C09150=1155.735,302.900,-72.976,-176.899,8.332,148.732
C09151=1155.730,303.148,-73.007,-176.896,8.334,148.732
C09152=1155.726,303.397,-73.038,-176.894,8.338,148.732
C09153=1155.722,303.644,-73.070,-176.892,8.341,148.732
C09154=1155.717,303.892,-73.100,-176.889,8.344,148.732
C09155=1155.713,304.141,-73.132,-176.887,8.347,148.732
C09156=1155.709,304.389,-73.162,-176.883,8.351,148.732
C09157=1155.705,304.636,-73.193,-176.881,8.354,148.733
C09158=1155.701,304.885,-73.224,-176.878,8.357,148.733
C09159=1155.696,305.132,-73.255,-176.876,8.361,148.733
C09160=1155.692,305.381,-73.286,-176.874,8.364,148.733
C09161=1155.688,305.628,-73.318,-176.870,8.368,148.733
C09162=1155.683,305.876,-73.349,-176.868,8.371,148.733
C09163=1155.679,306.125,-73.380,-176.865,8.374,148.733
C09164=1155.675,306.373,-73.410,-176.863,8.377,148.733
C09165=1155.672,306.621,-73.442,-176.861,8.380,148.734
C09166=1155.667,306.869,-73.472,-176.858,8.383,148.733
C09167=1155.663,307.117,-73.504,-176.855,8.387,148.734
C09168=1155.659,307.365,-73.535,-176.852,8.390,148.734
C09169=1155.654,307.613,-73.566,-176.850,8.394,148.734
C09170=1155.650,307.861,-73.598,-176.848,8.397,148.734
C09171=1155.646,308.109,-73.628,-176.845,8.400,148.734
C09172=1155.642,308.357,-73.660,-176.842,8.404,148.734
C09173=1155.638,308.605,-73.691,-176.840,8.407,148.734
C09174=1155.634,308.853,-73.722,-176.837,8.410,148.734
C09175=1155.629,309.101,-73.754,-176.835,8.414,148.735
C09176=1155.625,309.349,-73.785,-176.832,8.416,148.735
C09177=1155.621,309.597,-73.816,-176.829,8.421,148.735
C09178=1155.617,309.845,-73.847,-176.827,8.424,148.735
C09179=1155.613,310.093,-73.879,-176.824,8.427,148.735
C09180=1155.609,310.341,-73.911,-176.822,8.430,148.735
C09181=1155.604,310.589,-73.941,-176.819,8.433,148.735
C09182=1155.601,310.837,-73.973,-176.816,8.437,148.735
C09183=1155.596,311.085,-74.004,-176.814,8.440,148.736
C09184=1155.592,311.333,-74.036,-176.811,8.444,148.736
C09185=1155.587,311.580,-74.068,-176.809,8.447,148.736
C09186=1155.583,311.829,-74.099,-176.806,8.451,148.736
C09187=1155.579,312.077,-74.131,-176.803,8.454,148.736
C09188=1155.575,312.325,-74.162,-176.801,8.457,148.736
C09189=1155.571,312.573,-74.194,-176.798,8.460,148.736
C09190=1155.567,312.820,-74.225,-176.796,8.464,148.736
C09191=1155.563,313.068,-74.257,-176.793,8.467,148.737
C09192=1155.558,313.346,-74.291,-176.790,8.471,148.737
C09193=1155.554,313.623,-74.327,-176.788,8.475,148.737
C09194=1155.549,313.901,-74.363,-176.784,8.478,148.737
C09195=1155.544,314.178,-74.398,-176.781,8.483,148.737
C09196=1155.540,314.426,-74.430,-176.779,8.486,148.737
C09197=1155.535,314.674,-74.461,-176.777,8.489,148.738
C09198=1155.532,314.922,-74.493,-176.774,8.492,148.738
C09199=1155.528,315.170,-74.525,-176.771,8.496,148.738
C09200=1155.523,315.418,-74.557,-176.769,8.499,148.738
C09201=1155.519,315.666,-74.589,-176.766,8.502,148.738
C09202=1155.515,315.914,-74.621,-176.764,8.506,148.738
C09203=1155.511,316.162,-74.651,-176.761,8.510,148.738
C09204=1155.506,316.410,-74.684,-176.758,8.513,148.739
C09205=1155.503,316.658,-74.716,-176.756,8.516,148.739
C09206=1155.498,316.906,-74.747,-176.753,8.519,148.739
C09207=1155.495,317.154,-74.779,-176.750,8.523,148.739
C09208=1155.490,317.402,-74.811,-176.748,8.527,148.739
C09209=1155.486,317.649,-74.843,-176.745,8.530,148.739
C09210=1155.482,317.897,-74.875,-176.743,8.533,148.739
C09211=1155.478,318.146,-74.907,-176.740,8.537,148.740
C09212=1155.473,318.393,-74.939,-176.738,8.540,148.740
C09213=1155.470,318.641,-74.970,-176.735,8.543,148.740
C09214=1155.465,318.889,-75.003,-176.733,8.547,148.740
C09215=1155.461,319.137,-75.034,-176.730,8.551,148.740
C09216=1155.457,319.385,-75.066,-176.728,8.554,148.740
C09217=1155.453,319.633,-75.099,-176.725,8.557,148.740
C09218=1155.449,319.881,-75.131,-176.723,8.560,148.741
C09219=1155.445,320.129,-75.162,-176.720,8.564,148.741
C09220=1155.441,320.376,-75.195,-176.717,8.568,148.741
C09221=1155.437,320.624,-75.227,-176.715,8.571,148.741
C09222=1155.433,320.873,-75.259,-176.712,8.575,148.741
C09223=1155.428,321.120,-75.291,-176.709,8.578,148.741
C09224=1155.425,321.368,-75.323,-176.707,8.581,148.742
C09225=1155.420,321.616,-75.355,-176.705,8.584,148.742
C09226=1155.417,321.864,-75.388,-176.702,8.589,148.742
C09227=1155.412,322.111,-75.420,-176.699,8.592,148.742
C09228=1155.408,322.359,-75.452,-176.697,8.595,148.742
C09229=1155.403,322.608,-75.484,-176.694,8.599,148.742
C09230=1155.400,322.855,-75.517,-176.692,8.602,148.743
C09231=1155.396,323.104,-75.549,-176.689,8.605,148.743
C09232=1155.391,323.351,-75.581,-176.687,8.609,148.743
C09233=1155.387,323.599,-75.613,-176.684,8.612,148.743
C09234=1155.383,323.847,-75.646,-176.681,8.616,148.743
C09235=1155.379,324.095,-75.678,-176.679,8.619,148.743
C09236=1155.375,324.343,-75.710,-176.676,8.623,148.744
C09237=1155.371,324.590,-75.743,-176.674,8.626,148.744
C09238=1155.367,324.838,-75.775,-176.672,8.630,148.744
C09239=1155.363,325.086,-75.808,-176.669,8.633,148.744
C09240=1155.359,325.334,-75.840,-176.666,8.637,148.744
C09241=1155.355,325.582,-75.872,-176.664,8.640,148.744
C09242=1155.350,325.830,-75.905,-176.661,8.643,148.745
C09243=1155.347,326.078,-75.937,-176.658,8.647,148.745
C09244=1155.342,326.325,-75.970,-176.656,8.651,148.745
C09245=1155.338,326.573,-76.002,-176.654,8.654,148.745
C09246=1155.334,326.821,-76.035,-176.651,8.658,148.745
C09247=1155.330,327.069,-76.067,-176.648,8.661,148.745
C09248=1155.326,327.317,-76.100,-176.646,8.664,148.746
C09249=1155.322,327.565,-76.132,-176.643,8.668,148.746
C09250=1155.318,327.813,-76.165,-176.641,8.672,148.746
C09251=1155.314,328.061,-76.197,-176.638,8.675,148.746
C09252=1155.309,328.308,-76.230,-176.635,8.679,148.747
C09253=1155.305,328.556,-76.262,-176.633,8.682,148.747
C09254=1155.301,328.803,-76.295,-176.631,8.686,148.747
C09255=1155.297,329.051,-76.328,-176.628,8.690,148.747
C09256=1155.293,329.300,-76.361,-176.626,8.693,148.747
C09257=1155.289,329.547,-76.394,-176.623,8.696,148.747
C09258=1155.285,329.795,-76.426,-176.620,8.700,148.748
C09259=1155.281,330.043,-76.459,-176.618,8.703,148.748
C09260=1155.277,330.291,-76.492,-176.615,8.707,148.748
C09261=1155.273,330.539,-76.525,-176.612,8.711,148.748
C09262=1155.269,330.787,-76.557,-176.610,8.714,148.748
C09263=1155.265,331.034,-76.590,-176.608,8.717,148.749
C09264=1155.261,331.282,-76.623,-176.605,8.721,148.749
C09265=1155.257,331.530,-76.656,-176.603,8.725,148.749
C09266=1155.252,331.778,-76.689,-176.600,8.728,148.749
C09267=1155.249,332.026,-76.721,-176.597,8.732,148.750
C09268=1155.245,332.273,-76.755,-176.595,8.735,148.750
C09269=1155.240,332.521,-76.788,-176.593,8.739,148.750
C09270=1155.236,332.769,-76.821,-176.590,8.743,148.750
C09271=1155.232,333.017,-76.853,-176.587,8.746,148.750
C09272=1155.228,333.265,-76.886,-176.585,8.749,148.751
C09273=1155.224,333.513,-76.920,-176.582,8.753,148.751
C09274=1155.220,333.760,-76.952,-176.580,8.757,148.751
C09275=1155.216,334.008,-76.985,-176.578,8.760,148.751
C09276=1155.212,334.255,-77.018,-176.575,8.764,148.751
C09277=1155.208,334.503,-77.052,-176.572,8.767,148.752
C09278=1155.204,334.751,-77.085,-176.570,8.771,148.752
C09279=1155.199,334.999,-77.118,-176.567,8.775,148.752
C09280=1155.195,335.246,-77.151,-176.565,8.778,148.752
C09281=1155.191,335.494,-77.184,-176.562,8.782,148.753
C09282=1155.187,335.742,-77.217,-176.560,8.785,148.753
C09283=1155.183,335.990,-77.251,-176.557,8.789,148.753
C09284=1155.179,336.237,-77.284,-176.555,8.793,148.753
C09285=1155.175,336.485,-77.317,-176.552,8.796,148.753
C09286=1155.170,336.733,-77.350,-176.549,8.800,148.754
C09287=1155.166,336.980,-77.383,-176.547,8.803,148.754
C09288=1155.163,337.229,-77.417,-176.545,8.807,148.754
C09289=1155.159,337.477,-77.450,-176.542,8.811,148.754
C09290=1155.155,337.724,-77.483,-176.539,8.814,148.755
C09291=1155.150,337.972,-77.516,-176.537,8.818,148.755
C09292=1155.146,338.220,-77.549,-176.534,8.821,148.755
C09293=1155.142,338.468,-77.582,-176.532,8.825,148.755
C09294=1155.138,338.715,-77.616,-176.529,8.829,148.755
C09295=1155.134,338.962,-77.649,-176.527,8.832,148.756
C09296=1155.130,339.243,-77.687,-176.524,8.836,148.756
C09297=1155.126,339.522,-77.725,-176.521,8.840,148.756
C09298=1155.121,339.803,-77.763,-176.518,8.844,148.756
C09299=1155.116,340.082,-77.801,-176.515,8.848,148.757
C09300=1155.112,340.330,-77.834,-176.513,8.852,148.757
C09301=1155.108,340.578,-77.867,-176.510,8.856,148.757
C09302=1155.104,340.826,-77.900,-176.508,8.859,148.757
C09303=1155.101,341.073,-77.935,-176.505,8.863,148.758
C09304=1155.096,341.321,-77.968,-176.503,8.867,148.758
C09305=1155.092,341.569,-78.002,-176.501,8.870,148.758
C09306=1155.088,341.816,-78.035,-176.498,8.874,148.758
C09307=1155.084,342.064,-78.069,-176.495,8.877,148.759
C09308=1155.079,342.312,-78.102,-176.492,8.882,148.759
C09309=1155.075,342.560,-78.137,-176.490,8.885,148.759
C09310=1155.071,342.808,-78.170,-176.487,8.889,148.759
C09311=1155.067,343.055,-78.204,-176.485,8.892,148.760
C09312=1155.063,343.302,-78.237,-176.483,8.896,148.760
C09313=1155.059,343.551,-78.271,-176.480,8.900,148.760
C09314=1155.055,343.798,-78.305,-176.478,8.903,148.760
C09315=1155.051,344.046,-78.338,-176.475,8.907,148.761
C09316=1155.047,344.293,-78.372,-176.473,8.911,148.761
C09317=1155.042,344.541,-78.406,-176.470,8.915,148.761
C09318=1155.039,344.789,-78.440,-176.467,8.918,148.761
C09319=1155.035,345.037,-78.473,-176.466,8.921,148.762
C09320=1155.030,345.284,-78.507,-176.463,8.926,148.762
C09321=1155.027,345.532,-78.542,-176.460,8.929,148.762
C09322=1155.023,345.780,-78.575,-176.457,8.933,148.762
C09323=1155.019,346.027,-78.609,-176.455,8.936,148.763
C09324=1155.014,346.275,-78.642,-176.452,8.940,148.763
C09325=1155.011,346.523,-78.677,-176.450,8.944,148.763
C09326=1155.007,346.770,-78.711,-176.447,8.948,148.764
C09327=1155.002,347.018,-78.744,-176.445,8.951,148.764
C09328=1154.999,347.266,-78.778,-176.442,8.955,148.764
C09329=1154.995,347.513,-78.813,-176.440,8.959,148.764
C09330=1154.991,347.761,-78.846,-176.438,8.962,148.764
C09331=1154.987,348.009,-78.880,-176.435,8.966,148.765
C09332=1154.983,348.256,-78.915,-176.433,8.970,148.765
C09333=1154.979,348.504,-78.948,-176.430,8.974,148.765
C09334=1154.975,348.752,-78.983,-176.428,8.977,148.766
C09335=1154.971,348.999,-79.017,-176.425,8.981,148.766
C09336=1154.966,349.246,-79.051,-176.423,8.985,148.766
C09337=1154.963,349.494,-79.085,-176.420,8.989,148.766
C09338=1154.959,349.742,-79.119,-176.418,8.992,148.767
C09339=1154.954,349.989,-79.153,-176.415,8.996,148.767
C09340=1154.951,350.237,-79.187,-176.412,8.999,148.767
C09341=1154.946,350.485,-79.222,-176.410,9.004,148.768
C09342=1154.943,350.732,-79.256,-176.408,9.007,148.768
C09343=1154.939,350.980,-79.290,-176.405,9.011,148.768
C09344=1154.935,351.227,-79.324,-176.402,9.015,148.768
C09345=1154.931,351.476,-79.358,-176.400,9.019,148.769
C09346=1154.927,351.723,-79.392,-176.398,9.022,148.769
C09347=1154.923,351.971,-79.427,-176.395,9.026,148.769
C09348=1154.918,352.218,-79.462,-176.393,9.030,148.769
C09349=1154.914,352.465,-79.495,-176.390,9.034,148.770
C09350=1154.910,352.713,-79.530,-176.388,9.037,148.770
C09351=1154.907,352.961,-79.564,-176.385,9.041,148.770
C09352=1154.903,353.209,-79.599,-176.383,9.045,148.771
C09353=1154.899,353.456,-79.633,-176.380,9.049,148.771
C09354=1154.895,353.704,-79.668,-176.378,9.052,148.771
C09355=1154.890,353.951,-79.702,-176.375,9.056,148.772
C09356=1154.887,354.199,-79.736,-176.373,9.060,148.772
C09357=1154.882,354.447,-79.771,-176.370,9.064,148.772
C09358=1154.879,354.694,-79.806,-176.368,9.067,148.772
C09359=1154.875,354.941,-79.840,-176.365,9.071,148.773
C09360=1154.871,355.189,-79.875,-176.363,9.075,148.773
C09361=1154.867,355.436,-79.909,-176.360,9.079,148.773
C09362=1154.863,355.685,-79.944,-176.358,9.082,148.774
C09363=1154.859,355.932,-79.978,-176.355,9.087,148.774
C09364=1154.855,356.180,-80.013,-176.353,9.090,148.774
C09365=1154.851,356.427,-80.048,-176.350,9.094,148.775
C09366=1154.847,356.675,-80.083,-176.348,9.098,148.775
C09367=1154.843,356.922,-80.116,-176.345,9.102,148.775
C09368=1154.839,357.170,-80.151,-176.343,9.105,148.775
C09369=1154.835,357.417,-80.186,-176.341,9.110,148.776
C09370=1154.831,357.665,-80.221,-176.338,9.113,148.776
C09371=1154.827,357.912,-80.255,-176.335,9.117,148.776
C09372=1154.824,358.159,-80.291,-176.333,9.121,148.777
C09373=1154.819,358.407,-80.325,-176.331,9.125,148.777
C09374=1154.815,358.655,-80.360,-176.328,9.129,148.777
C09375=1154.812,358.902,-80.395,-176.326,9.132,148.778
C09376=1154.808,359.150,-80.429,-176.323,9.136,148.778
C09377=1154.804,359.398,-80.464,-176.321,9.140,148.778
C09378=1154.799,359.645,-80.499,-176.318,9.144,148.779
C09379=1154.795,359.893,-80.534,-176.315,9.148,148.779
C09380=1154.792,360.140,-80.568,-176.313,9.152,148.779
C09381=1154.788,360.387,-80.604,-176.310,9.156,148.780
C09382=1154.784,360.635,-80.638,-176.308,9.159,148.780
C09383=1154.780,360.882,-80.674,-176.305,9.163,148.780
C09384=1154.776,361.130,-80.708,-176.303,9.168,148.781
C09385=1154.772,361.378,-80.744,-176.300,9.171,148.781
C09386=1154.767,361.625,-80.779,-176.297,9.175,148.781
C09387=1154.765,361.872,-80.813,-176.295,9.179,148.781
C09388=1154.761,362.121,-80.848,-176.293,9.183,148.782
C09389=1154.756,362.367,-80.883,-176.290,9.187,148.782
C09390=1154.753,362.615,-80.919,-176.287,9.191,148.782
C09391=1154.749,362.863,-80.954,-176.285,9.195,148.783
C09392=1154.744,363.110,-80.989,-176.283,9.199,148.783
C09393=1154.740,363.358,-81.024,-176.280,9.202,148.783
C09394=1154.737,363.605,-81.059,-176.278,9.207,148.784
C09395=1154.732,363.852,-81.095,-176.275,9.211,148.784
C09396=1154.729,364.100,-81.129,-176.273,9.214,148.784
C09397=1154.725,364.348,-81.165,-176.270,9.218,148.785
C09398=1154.721,364.595,-81.201,-176.267,9.223,148.785
C09399=1154.717,364.843,-81.235,-176.265,9.226,148.785
C09400=1154.713,365.126,-81.275,-176.262,9.231,148.786
C09401=1154.708,365.408,-81.316,-176.259,9.235,148.786
C09402=1154.703,365.692,-81.356,-176.257,9.240,148.787
C09403=1154.699,365.974,-81.396,-176.253,9.245,148.787
C09404=1154.696,366.222,-81.432,-176.252,9.248,148.787
C09405=1154.692,366.469,-81.467,-176.249,9.252,148.788
C09406=1154.688,366.716,-81.502,-176.246,9.257,148.788
C09407=1154.683,366.964,-81.538,-176.244,9.260,148.788
C09408=1154.679,367.212,-81.573,-176.241,9.265,148.789
C09409=1154.676,367.459,-81.609,-176.239,9.269,148.789
C09410=1154.671,367.706,-81.644,-176.237,9.272,148.790
C09411=1154.668,367.954,-81.680,-176.234,9.277,148.790
C09412=1154.664,368.201,-81.715,-176.232,9.280,148.790
C09413=1154.660,368.449,-81.751,-176.229,9.284,148.791
C09414=1154.657,368.696,-81.786,-176.227,9.289,148.791
C09415=1154.652,368.943,-81.822,-176.225,9.292,148.792
C09416=1154.648,369.191,-81.858,-176.223,9.297,148.792
C09417=1154.644,369.438,-81.893,-176.220,9.301,148.792
C09418=1154.641,369.686,-81.929,-176.218,9.304,148.793
C09419=1154.637,369.933,-81.964,-176.215,9.309,148.793
C09420=1154.633,370.180,-82.000,-176.213,9.312,148.794
C09421=1154.628,370.428,-82.036,-176.211,9.317,148.794
C09422=1154.625,370.675,-82.071,-176.208,9.321,148.795
C09423=1154.621,370.923,-82.107,-176.207,9.325,148.795
C09424=1154.617,371.170,-82.142,-176.204,9.329,148.796
C09425=1154.613,371.418,-82.178,-176.202,9.333,148.796
C09426=1154.609,371.666,-82.214,-176.200,9.337,148.796
C09427=1154.605,371.913,-82.249,-176.198,9.341,148.797
C09428=1154.601,372.160,-82.285,-176.195,9.345,148.797
C09429=1154.597,372.407,-82.322,-176.193,9.349,148.798
C09430=1154.594,372.655,-82.357,-176.191,9.353,148.798
C09431=1154.590,372.902,-82.393,-176.189,9.357,148.799
C09432=1154.586,373.150,-82.428,-176.187,9.361,148.799
C09433=1154.582,373.398,-82.464,-176.185,9.365,148.800
C09434=1154.579,373.644,-82.501,-176.183,9.369,148.800
C09435=1154.574,373.891,-82.536,-176.181,9.373,148.801
C09436=1154.570,374.139,-82.572,-176.179,9.378,148.801
C09437=1154.566,374.387,-82.608,-176.177,9.381,148.802
C09438=1154.563,374.633,-82.644,-176.175,9.385,148.802
C09439=1154.558,374.881,-82.680,-176.173,9.390,148.803
C09440=1154.555,375.129,-82.715,-176.171,9.393,148.803
C09441=1154.551,375.376,-82.751,-176.170,9.397,148.804
C09442=1154.547,375.623,-82.788,-176.167,9.401,148.804
C09443=1154.543,375.871,-82.823,-176.166,9.405,148.805
C09444=1154.539,376.118,-82.860,-176.164,9.409,148.806
C09445=1154.536,376.366,-82.896,-176.162,9.414,148.806
C09446=1154.532,376.613,-82.931,-176.160,9.418,148.807
C09447=1154.528,376.860,-82.968,-176.159,9.421,148.807
C09448=1154.524,377.108,-83.004,-176.157,9.425,148.808
C09449=1154.520,377.356,-83.040,-176.155,9.429,148.808
C09450=1154.516,377.602,-83.076,-176.154,9.433,148.809
C09451=1154.512,377.850,-83.112,-176.152,9.438,148.810
C09452=1154.509,378.097,-83.149,-176.150,9.441,148.810
C09453=1154.504,378.345,-83.185,-176.149,9.445,148.811
C09454=1154.501,378.592,-83.221,-176.148,9.449,148.812
C09455=1154.497,378.840,-83.257,-176.146,9.453,148.812
C09456=1154.493,379.087,-83.293,-176.145,9.457,148.813
C09457=1154.489,379.334,-83.330,-176.143,9.461,148.813
C09458=1154.485,379.581,-83.366,-176.142,9.465,148.814
C09459=1154.481,379.829,-83.402,-176.141,9.469,148.815
C09460=1154.478,380.076,-83.438,-176.140,9.472,148.815
C09461=1154.473,380.324,-83.474,-176.138,9.476,148.816
C09462=1154.470,380.571,-83.511,-176.137,9.480,148.817
C09463=1154.466,380.818,-83.547,-176.136,9.484,148.817
C09464=1154.462,381.065,-83.583,-176.135,9.488,148.818
C09465=1154.458,381.313,-83.620,-176.134,9.491,148.819
C09466=1154.454,381.560,-83.655,-176.133,9.496,148.820
C09467=1154.450,381.807,-83.692,-176.131,9.499,148.820
C09468=1154.447,382.054,-83.729,-176.131,9.503,148.821
C09469=1154.443,382.302,-83.765,-176.130,9.507,148.822
C09470=1154.438,382.549,-83.802,-176.129,9.510,148.822
C09471=1154.435,382.796,-83.838,-176.128,9.514,148.823
C09472=1154.431,383.044,-83.874,-176.127,9.518,148.824
C09473=1154.427,383.291,-83.910,-176.127,9.521,148.825
C09474=1154.423,383.538,-83.947,-176.126,9.525,148.825
C09475=1154.419,383.786,-83.983,-176.125,9.528,148.826
C09476=1154.415,384.033,-84.019,-176.125,9.532,148.827
C09477=1154.411,384.280,-84.056,-176.124,9.535,148.828
C09478=1154.408,384.527,-84.092,-176.123,9.539,148.828
C09479=1154.404,384.774,-84.129,-176.123,9.543,148.829
C09480=1154.400,385.022,-84.166,-176.123,9.546,148.830
C09481=1154.397,385.269,-84.202,-176.122,9.550,148.831
C09482=1154.392,385.517,-84.238,-176.122,9.553,148.832
C09483=1154.388,385.764,-84.275,-176.122,9.556,148.832
C09484=1154.385,386.011,-84.311,-176.121,9.559,148.833
C09485=1154.381,386.258,-84.348,-176.121,9.563,148.834
C09486=1154.377,386.505,-84.385,-176.121,9.566,148.835
C09487=1154.373,386.753,-84.421,-176.121,9.569,148.836
C09488=1154.369,387.000,-84.458,-176.121,9.572,148.837
C09489=1154.366,387.247,-84.494,-176.120,9.576,148.837
C09490=1154.362,387.495,-84.531,-176.121,9.579,148.838
C09491=1154.358,387.742,-84.568,-176.121,9.582,148.839
C09492=1154.354,387.990,-84.604,-176.121,9.585,148.840
C09493=1154.350,388.237,-84.640,-176.121,9.588,148.841
C09494=1154.346,388.484,-84.677,-176.121,9.591,148.842
C09495=1154.343,388.731,-84.713,-176.121,9.594,148.842
C09496=1154.339,388.978,-84.750,-176.122,9.597,148.843
C09497=1154.334,389.226,-84.786,-176.122,9.600,148.844
C09498=1154.332,389.473,-84.823,-176.122,9.603,148.845
C09499=1154.327,389.721,-84.860,-176.122,9.606,148.846
C09500=1154.323,389.968,-84.897,-176.123,9.608,148.846
C09501=1154.319,390.215,-84.934,-176.123,9.611,148.847
C09502=1154.316,390.462,-84.970,-176.124,9.614,148.848
C09503=1154.312,390.709,-85.007,-176.124,9.617,148.849
C09504=1154.307,390.996,-85.049,-176.125,9.620,148.850
C09505=1154.302,391.282,-85.091,-176.125,9.623,148.851
C09506=1154.299,391.568,-85.134,-176.125,9.626,148.852
C09507=1154.294,391.854,-85.176,-176.126,9.630,148.853
C09508=1154.291,392.102,-85.213,-176.127,9.632,148.854
C09509=1154.286,392.349,-85.250,-176.127,9.634,148.855
C09510=1154.283,392.596,-85.286,-176.128,9.637,148.855
C09511=1154.279,392.843,-85.323,-176.129,9.640,148.856
C09512=1154.275,393.090,-85.360,-176.130,9.642,148.857
C09513=1154.271,393.337,-85.397,-176.130,9.645,148.858
C09514=1154.267,393.584,-85.433,-176.130,9.647,148.859
C09515=1154.264,393.833,-85.469,-176.131,9.650,148.860
C09516=1154.260,394.080,-85.506,-176.132,9.652,148.861
C09517=1154.255,394.327,-85.543,-176.133,9.654,148.861
C09518=1154.252,394.574,-85.579,-176.133,9.657,148.862
C09519=1154.248,394.821,-85.616,-176.134,9.660,148.863
C09520=1154.244,395.068,-85.653,-176.135,9.662,148.864
C09521=1154.240,395.316,-85.690,-176.136,9.664,148.864
C09522=1154.237,395.563,-85.727,-176.136,9.667,148.865
C09523=1154.233,395.810,-85.763,-176.137,9.669,148.866
C09524=1154.229,396.058,-85.800,-176.138,9.672,148.867
C09525=1154.226,396.304,-85.836,-176.139,9.674,148.868
C09526=1154.221,396.552,-85.873,-176.140,9.675,148.869
C09527=1154.217,396.799,-85.909,-176.140,9.678,148.869
C09528=1154.213,397.047,-85.946,-176.141,9.680,148.870
C09529=1154.210,397.294,-85.983,-176.142,9.682,148.871
C09530=1154.206,397.541,-86.020,-176.142,9.685,148.872
C09531=1154.202,397.789,-86.057,-176.144,9.687,148.873
C09532=1154.198,398.036,-86.094,-176.145,9.689,148.874
C09533=1154.194,398.283,-86.130,-176.145,9.691,148.874
C09534=1154.190,398.530,-86.167,-176.146,9.693,148.875
C09535=1154.187,398.778,-86.204,-176.147,9.696,148.876
C09536=1154.183,399.025,-86.241,-176.148,9.697,148.877
C09537=1154.179,399.272,-86.278,-176.149,9.700,148.877
C09538=1154.175,399.519,-86.314,-176.150,9.702,148.878
C09539=1154.171,399.766,-86.351,-176.151,9.703,148.879
C09540=1154.167,400.013,-86.388,-176.152,9.705,148.880
C09541=1154.163,400.261,-86.424,-176.152,9.708,148.881
C09542=1154.160,400.508,-86.461,-176.153,9.710,148.881
C09543=1154.156,400.756,-86.497,-176.154,9.712,148.882
C09544=1154.152,401.003,-86.534,-176.155,9.714,148.883
C09545=1154.148,401.250,-86.571,-176.156,9.716,148.884
C09546=1154.144,401.497,-86.607,-176.157,9.718,148.884
C09547=1154.140,401.744,-86.644,-176.158,9.720,148.885
C09548=1154.137,401.992,-86.681,-176.159,9.722,148.886
C09549=1154.133,402.239,-86.718,-176.160,9.723,148.887
C09550=1154.129,402.486,-86.754,-176.161,9.726,148.887
C09551=1154.125,402.734,-86.791,-176.161,9.727,148.888
C09552=1154.121,402.981,-86.828,-176.162,9.729,148.889
C09553=1154.117,403.228,-86.865,-176.163,9.731,148.890
C09554=1154.114,403.475,-86.901,-176.164,9.733,148.890
C09555=1154.110,403.723,-86.938,-176.165,9.735,148.891
C09556=1154.106,403.970,-86.975,-176.166,9.737,148.892
C09557=1154.102,404.217,-87.012,-176.167,9.739,148.893
C09558=1154.098,404.464,-87.049,-176.167,9.740,148.893
C09559=1154.095,404.711,-87.085,-176.169,9.743,148.894
C09560=1154.091,404.958,-87.122,-176.169,9.744,148.895
C09561=1154.087,405.206,-87.159,-176.170,9.746,148.895
C09562=1154.083,405.453,-87.196,-176.171,9.748,148.896
C09563=1154.080,405.700,-87.233,-176.172,9.750,148.897
C09564=1154.076,405.947,-87.269,-176.173,9.752,148.898
C09565=1154.071,406.195,-87.306,-176.173,9.754,148.898
C09566=1154.067,406.442,-87.342,-176.174,9.755,148.899
C09567=1154.064,406.690,-87.379,-176.175,9.757,148.900
C09568=1154.060,406.937,-87.416,-176.176,9.759,148.900
C09569=1154.056,407.184,-87.453,-176.177,9.761,148.901
C09570=1154.052,407.432,-87.490,-176.178,9.763,148.902
C09571=1154.048,407.679,-87.526,-176.178,9.765,148.903
C09572=1154.045,407.926,-87.563,-176.179,9.767,148.903
C09573=1154.041,408.174,-87.600,-176.180,9.768,148.904
C09574=1154.037,408.421,-87.637,-176.181,9.770,148.904
C09575=1154.033,408.668,-87.674,-176.182,9.772,148.905
C09576=1154.029,408.915,-87.710,-176.182,9.774,148.906
C09577=1154.025,409.162,-87.747,-176.183,9.776,148.907
C09578=1154.021,409.409,-87.784,-176.183,9.778,148.907
C09579=1154.018,409.657,-87.821,-176.184,9.780,148.908
C09580=1154.014,409.904,-87.857,-176.185,9.782,148.909
C09581=1154.010,410.151,-87.894,-176.186,9.784,148.909
C09582=1154.006,410.398,-87.931,-176.186,9.785,148.910
C09583=1154.002,410.646,-87.968,-176.187,9.787,148.911
C09584=1153.998,410.893,-88.005,-176.188,9.789,148.911
C09585=1153.995,411.140,-88.041,-176.188,9.791,148.912
C09586=1153.991,411.388,-88.078,-176.189,9.792,148.913
C09587=1153.987,411.635,-88.115,-176.190,9.794,148.913
C09588=1153.983,411.882,-88.152,-176.190,9.796,148.914
C09589=1153.979,412.129,-88.189,-176.191,9.798,148.915
C09590=1153.976,412.376,-88.225,-176.192,9.799,148.915
C09591=1153.971,412.623,-88.262,-176.192,9.801,148.916
C09592=1153.968,412.871,-88.299,-176.193,9.803,148.916
C09593=1153.964,413.118,-88.336,-176.194,9.805,148.917
C09594=1153.960,413.365,-88.373,-176.195,9.807,148.918
C09595=1153.956,413.612,-88.409,-176.195,9.809,148.919
C09596=1153.952,413.860,-88.446,-176.195,9.811,148.919
C09597=1153.948,414.107,-88.483,-176.196,9.813,148.920
C09598=1153.945,414.355,-88.520,-176.197,9.814,148.920
C09599=1153.941,414.601,-88.556,-176.197,9.816,148.921
C09600=1153.937,414.849,-88.593,-176.198,9.818,148.922
C09601=1153.934,415.097,-88.630,-176.199,9.820,148.922
C09602=1153.931,415.343,-88.666,-176.199,9.821,148.923
C09603=1153.929,415.591,-88.704,-176.199,9.824,148.924
C09604=1153.928,416.003,-88.764,-176.201,9.826,148.925
C09605=1153.929,416.415,-88.824,-176.201,9.829,148.926
C09606=1153.933,416.828,-88.885,-176.202,9.832,148.927
C09607=1153.938,417.239,-88.945,-176.203,9.835,148.928
C09608=1153.517,417.241,-88.993,-176.206,9.846,148.931
C09609=1153.512,416.826,-88.932,-176.205,9.843,148.930
C09610=1153.508,416.411,-88.871,-176.204,9.841,148.929
C09611=1153.507,415.995,-88.810,-176.203,9.838,148.928
C09612=1153.509,415.578,-88.749,-176.202,9.835,148.927
C09613=1153.511,415.332,-88.712,-176.201,9.833,148.926
C09614=1153.513,415.084,-88.676,-176.201,9.831,148.926
C09615=1153.517,414.837,-88.640,-176.201,9.828,148.925
C09616=1153.520,414.589,-88.602,-176.200,9.827,148.925
C09617=1153.524,414.342,-88.565,-176.199,9.825,148.924
C09618=1153.528,414.095,-88.529,-176.199,9.824,148.923
C09619=1153.532,413.848,-88.492,-176.198,9.822,148.923
C09620=1153.536,413.601,-88.455,-176.198,9.820,148.922
C09621=1153.540,413.354,-88.419,-176.197,9.818,148.921
C09622=1153.543,413.106,-88.381,-176.196,9.816,148.921
C09623=1153.547,412.859,-88.345,-176.196,9.814,148.920
C09624=1153.551,412.612,-88.308,-176.195,9.812,148.919
C09625=1153.555,412.365,-88.271,-176.194,9.810,148.919
C09626=1153.559,412.117,-88.235,-176.194,9.808,148.918
C09627=1153.563,411.870,-88.198,-176.193,9.807,148.917
C09628=1153.566,411.623,-88.161,-176.192,9.805,148.917
C09629=1153.570,411.375,-88.124,-176.192,9.803,148.916
C09630=1153.574,411.128,-88.087,-176.191,9.801,148.915
C09631=1153.578,410.881,-88.050,-176.190,9.800,148.915
C09632=1153.582,410.634,-88.014,-176.190,9.798,148.914
C09633=1153.586,410.387,-87.977,-176.189,9.796,148.914
C09634=1153.589,410.139,-87.940,-176.188,9.794,148.913
C09635=1153.593,409.892,-87.903,-176.187,9.792,148.912
C09636=1153.597,409.645,-87.866,-176.186,9.791,148.911
C09637=1153.601,409.398,-87.830,-176.186,9.789,148.911
C09638=1153.605,409.151,-87.793,-176.185,9.787,148.910
C09639=1153.609,408.904,-87.756,-176.184,9.785,148.909
C09640=1153.612,408.656,-87.719,-176.183,9.783,148.909
C09641=1153.616,408.408,-87.682,-176.183,9.782,148.908
C09642=1153.620,408.162,-87.646,-176.182,9.780,148.907
C09643=1153.624,407.914,-87.609,-176.181,9.778,148.907
C09644=1153.628,407.667,-87.572,-176.180,9.776,148.906
C09645=1153.632,407.420,-87.536,-176.179,9.774,148.905
C09646=1153.635,407.172,-87.499,-176.179,9.772,148.905
C09647=1153.639,406.925,-87.462,-176.178,9.770,148.904
C09648=1153.643,406.678,-87.425,-176.177,9.769,148.903
C09649=1153.647,406.431,-87.388,-176.176,9.767,148.902
C09650=1153.651,406.184,-87.351,-176.175,9.765,148.902
C09651=1153.655,405.937,-87.315,-176.174,9.763,148.901
C09652=1153.658,405.689,-87.278,-176.174,9.761,148.900
C09653=1153.662,405.442,-87.241,-176.173,9.759,148.900
C09654=1153.666,405.194,-87.204,-176.172,9.758,148.899
C09655=1153.670,404.948,-87.168,-176.171,9.756,148.898
C09656=1153.674,404.700,-87.131,-176.170,9.754,148.897
C09657=1153.678,404.453,-87.094,-176.170,9.752,148.897
C09658=1153.681,404.205,-87.057,-176.168,9.750,148.896
C09659=1153.685,403.958,-87.020,-176.168,9.748,148.895
C09660=1153.689,403.711,-86.984,-176.167,9.746,148.894
C09661=1153.693,403.464,-86.947,-176.166,9.744,148.894
C09662=1153.697,403.217,-86.910,-176.165,9.742,148.893
C09663=1153.701,402.970,-86.873,-176.164,9.741,148.892
C09664=1153.704,402.722,-86.837,-176.163,9.738,148.891
C09665=1153.708,402.475,-86.800,-176.162,9.737,148.891
C09666=1153.712,402.228,-86.763,-176.161,9.735,148.890
C09667=1153.716,401.981,-86.726,-176.161,9.733,148.889
C09668=1153.719,401.734,-86.690,-176.159,9.731,148.888
C09669=1153.724,401.486,-86.653,-176.159,9.729,148.888
C09670=1153.727,401.239,-86.616,-176.158,9.727,148.887
C09671=1153.731,400.991,-86.579,-176.157,9.724,148.886
C09672=1153.735,400.744,-86.542,-176.156,9.722,148.885
C09673=1153.739,400.497,-86.507,-176.155,9.720,148.885
C09674=1153.743,400.249,-86.470,-176.155,9.719,148.884
C09675=1153.747,400.002,-86.433,-176.153,9.717,148.883
C09676=1153.751,399.754,-86.396,-176.152,9.714,148.882
C09677=1153.754,399.508,-86.359,-176.152,9.713,148.882
C09678=1153.758,399.260,-86.322,-176.151,9.711,148.881
C09679=1153.762,399.013,-86.286,-176.149,9.709,148.880
C09680=1153.766,398.766,-86.249,-176.149,9.706,148.879
C09681=1153.770,398.519,-86.212,-176.148,9.704,148.878
C09682=1153.774,398.272,-86.176,-176.147,9.702,148.878
C09683=1153.777,398.024,-86.138,-176.146,9.700,148.877
C09684=1153.781,397.777,-86.102,-176.145,9.698,148.876
C09685=1153.785,397.530,-86.065,-176.145,9.695,148.875
C09686=1153.789,397.283,-86.028,-176.144,9.693,148.874
C09687=1153.793,397.036,-85.992,-176.142,9.691,148.874
C09688=1153.797,396.788,-85.955,-176.142,9.689,148.873
C09689=1153.800,396.540,-85.917,-176.141,9.687,148.872
C09690=1153.804,396.294,-85.881,-176.140,9.684,148.871
C09691=1153.808,396.046,-85.844,-176.139,9.682,148.870
C09692=1153.812,395.799,-85.807,-176.139,9.680,148.870
C09693=1153.816,395.551,-85.771,-176.138,9.678,148.869
C09694=1153.820,395.305,-85.735,-176.137,9.675,148.868
C09695=1153.824,395.057,-85.698,-176.136,9.673,148.867
C09696=1153.827,394.809,-85.661,-176.136,9.670,148.866
C09697=1153.831,394.562,-85.624,-176.135,9.668,148.865
C09698=1153.835,394.315,-85.588,-176.134,9.665,148.865
C09699=1153.839,394.068,-85.551,-176.133,9.663,148.864
C09700=1153.843,393.821,-85.514,-176.133,9.660,148.863
C09701=1153.847,393.574,-85.477,-176.132,9.659,148.862
C09702=1153.850,393.327,-85.441,-176.131,9.656,148.861
C09703=1153.854,393.079,-85.404,-176.130,9.654,148.860
C09704=1153.858,392.832,-85.367,-176.130,9.651,148.860
C09705=1153.861,392.585,-85.331,-176.129,9.648,148.859
C09706=1153.866,392.337,-85.295,-176.129,9.645,148.858
C09707=1153.870,392.090,-85.258,-176.128,9.643,148.857
C09708=1153.874,391.843,-85.221,-176.128,9.640,148.856
C09709=1153.877,391.557,-85.178,-176.127,9.638,148.855
C09710=1153.882,391.270,-85.136,-176.126,9.635,148.854
C09711=1153.887,390.984,-85.094,-176.126,9.631,148.853
C09712=1153.891,390.698,-85.051,-176.126,9.628,148.852
C09713=1153.895,390.451,-85.014,-176.125,9.625,148.851
C09714=1153.899,390.204,-84.977,-176.124,9.622,148.851
C09715=1153.902,389.957,-84.941,-176.124,9.620,148.850
C09716=1153.907,389.709,-84.905,-176.124,9.617,148.849
C09717=1153.911,389.462,-84.868,-176.123,9.614,148.848
C09718=1153.914,389.214,-84.831,-176.123,9.611,148.847
C09719=1153.918,388.967,-84.794,-176.123,9.608,148.846
C09720=1153.922,388.720,-84.758,-176.123,9.605,148.846
C09721=1153.925,388.473,-84.721,-176.123,9.602,148.845
C09722=1153.929,388.226,-84.685,-176.122,9.600,148.844
C09723=1153.934,387.978,-84.648,-176.122,9.596,148.843
C09724=1153.937,387.731,-84.612,-176.122,9.593,148.842
C09725=1153.941,387.484,-84.575,-176.122,9.590,148.841
C09726=1153.945,387.236,-84.538,-176.122,9.587,148.841
C09727=1153.948,386.989,-84.502,-176.122,9.583,148.840
C09728=1153.952,386.741,-84.466,-176.122,9.581,148.839
C09729=1153.956,386.494,-84.429,-176.122,9.577,148.838
C09730=1153.960,386.247,-84.392,-176.123,9.574,148.837
C09731=1153.964,386.000,-84.356,-176.123,9.571,148.837
C09732=1153.968,385.753,-84.319,-176.123,9.567,148.836
C09733=1153.972,385.505,-84.283,-176.123,9.564,148.835
C09734=1153.976,385.258,-84.246,-176.124,9.561,148.834
C09735=1153.979,385.010,-84.209,-176.124,9.557,148.833
C09736=1153.983,384.763,-84.173,-176.124,9.554,148.833
C09737=1153.987,384.515,-84.137,-176.125,9.551,148.832
C09738=1153.991,384.268,-84.100,-176.125,9.547,148.831
C09739=1153.994,384.021,-84.064,-176.126,9.544,148.830
C09740=1153.999,383.774,-84.027,-176.127,9.540,148.830
C09741=1154.002,383.527,-83.991,-176.127,9.536,148.829
C09742=1154.006,383.280,-83.954,-176.128,9.533,148.828
C09743=1154.010,383.032,-83.917,-176.129,9.529,148.827
C09744=1154.014,382.785,-83.882,-176.129,9.525,148.826
C09745=1154.018,382.538,-83.845,-176.130,9.521,148.826
C09746=1154.021,382.291,-83.809,-176.131,9.518,148.825
C09747=1154.026,382.043,-83.773,-176.132,9.514,148.824
C09748=1154.030,381.796,-83.736,-176.133,9.511,148.824
C09749=1154.033,381.548,-83.699,-176.134,9.506,148.823
C09750=1154.037,381.300,-83.663,-176.135,9.503,148.822
C09751=1154.040,381.053,-83.627,-176.136,9.499,148.821
C09752=1154.045,380.806,-83.590,-176.138,9.495,148.821
C09753=1154.048,380.559,-83.554,-176.139,9.491,148.820
C09754=1154.052,380.312,-83.518,-176.140,9.488,148.819
C09755=1154.056,380.064,-83.482,-176.141,9.484,148.819
C09756=1154.060,379.817,-83.445,-176.142,9.480,148.818
C09757=1154.063,379.570,-83.409,-176.143,9.476,148.817
C09758=1154.068,379.322,-83.373,-176.145,9.472,148.817
C09759=1154.071,379.075,-83.336,-176.146,9.468,148.816
C09760=1154.076,378.828,-83.300,-176.148,9.464,148.816
C09761=1154.079,378.581,-83.264,-176.149,9.460,148.815
C09762=1154.083,378.333,-83.228,-176.150,9.456,148.814
C09763=1154.087,378.086,-83.192,-176.152,9.452,148.813
C09764=1154.091,377.838,-83.155,-176.154,9.449,148.813
C09765=1154.094,377.591,-83.119,-176.155,9.445,148.812
C09766=1154.099,377.343,-83.083,-176.157,9.440,148.812
C09767=1154.103,377.096,-83.048,-176.159,9.436,148.811
C09768=1154.107,376.849,-83.011,-176.160,9.432,148.811
C09769=1154.110,376.601,-82.975,-176.162,9.429,148.810
C09770=1154.114,376.354,-82.938,-176.164,9.424,148.809
C09771=1154.118,376.107,-82.903,-176.166,9.420,148.809
C09772=1154.122,375.860,-82.868,-176.167,9.417,148.808
C09773=1154.126,375.613,-82.831,-176.169,9.413,148.808
C09774=1154.130,375.365,-82.795,-176.171,9.408,148.807
C09775=1154.134,375.117,-82.759,-176.173,9.404,148.807
C09776=1154.138,374.870,-82.723,-176.174,9.401,148.806
C09777=1154.141,374.623,-82.687,-176.177,9.396,148.806
C09778=1154.146,374.375,-82.651,-176.179,9.393,148.805
C09779=1154.149,374.128,-82.615,-176.181,9.388,148.805
C09780=1154.153,373.881,-82.579,-176.183,9.384,148.804
C09781=1154.157,373.633,-82.543,-176.185,9.380,148.804
C09782=1154.161,373.385,-82.508,-176.187,9.376,148.803
C09783=1154.164,373.139,-82.471,-176.189,9.372,148.803
C09784=1154.169,372.891,-82.435,-176.191,9.368,148.802
C09785=1154.173,372.644,-82.400,-176.193,9.364,148.802
C09786=1154.177,372.396,-82.364,-176.195,9.360,148.801
C09787=1154.180,372.149,-82.329,-176.198,9.356,148.801
C09788=1154.184,371.902,-82.292,-176.200,9.352,148.800
C09789=1154.188,371.654,-82.256,-176.202,9.348,148.800
C09790=1154.192,371.407,-82.221,-176.204,9.344,148.799
C09791=1154.195,371.159,-82.185,-176.206,9.340,148.799
C09792=1154.200,370.912,-82.150,-176.208,9.336,148.799
C09793=1154.204,370.665,-82.114,-176.211,9.332,148.798
C09794=1154.208,370.417,-82.078,-176.213,9.327,148.798
C09795=1154.211,370.170,-82.043,-176.215,9.324,148.797
C09796=1154.216,369.922,-82.007,-176.218,9.319,148.797
C09797=1154.219,369.674,-81.971,-176.220,9.316,148.796
C09798=1154.224,369.428,-81.936,-176.222,9.311,148.796
C09799=1154.227,369.180,-81.901,-176.225,9.307,148.796
C09800=1154.231,368.932,-81.865,-176.227,9.303,148.795
C09801=1154.235,368.685,-81.829,-176.229,9.299,148.795
C09802=1154.239,368.437,-81.793,-176.231,9.296,148.794
C09803=1154.243,368.190,-81.758,-176.234,9.291,148.794
C09804=1154.247,367.943,-81.723,-176.237,9.287,148.793
C09805=1154.251,367.695,-81.687,-176.238,9.283,148.793
C09806=1154.254,367.448,-81.651,-176.241,9.279,148.793
C09807=1154.258,367.200,-81.616,-176.244,9.275,148.792
C09808=1154.262,366.954,-81.581,-176.246,9.272,148.792
C09809=1154.266,366.705,-81.546,-176.249,9.267,148.792
C09810=1154.271,366.458,-81.510,-176.251,9.263,148.791
C09811=1154.274,366.210,-81.474,-176.253,9.260,148.791
C09812=1154.279,365.963,-81.439,-176.256,9.255,148.790
C09813=1154.282,365.680,-81.399,-176.259,9.251,148.790
C09814=1154.287,365.398,-81.358,-176.262,9.246,148.790
C09815=1154.292,365.114,-81.318,-176.265,9.242,148.789
C09816=1154.296,364.832,-81.278,-176.267,9.237,148.789
C09817=1154.300,364.584,-81.243,-176.270,9.233,148.788
C09818=1154.304,364.336,-81.207,-176.273,9.229,148.788
C09819=1154.307,364.089,-81.172,-176.275,9.226,148.788
C09820=1154.312,363.841,-81.137,-176.277,9.221,148.787
C09821=1154.316,363.594,-81.102,-176.280,9.217,148.787
C09822=1154.319,363.346,-81.066,-176.282,9.213,148.787
C09823=1154.324,363.099,-81.032,-176.285,9.209,148.787
C09824=1154.327,362.851,-80.996,-176.287,9.205,148.786
C09825=1154.331,362.604,-80.961,-176.290,9.202,148.786
C09826=1154.336,362.357,-80.926,-176.293,9.198,148.786
C09827=1154.339,362.109,-80.891,-176.295,9.193,148.785
C09828=1154.343,361.861,-80.856,-176.297,9.190,148.785
C09829=1154.347,361.614,-80.821,-176.300,9.186,148.785
C09830=1154.351,361.366,-80.786,-176.302,9.182,148.784
C09831=1154.354,361.119,-80.751,-176.305,9.178,148.784
C09832=1154.359,360.871,-80.716,-176.308,9.174,148.783
C09833=1154.363,360.624,-80.681,-176.310,9.170,148.783
C09834=1154.367,360.376,-80.646,-176.313,9.166,148.783
C09835=1154.371,360.129,-80.611,-176.315,9.162,148.783
C09836=1154.374,359.881,-80.577,-176.318,9.159,148.782
C09837=1154.378,359.634,-80.541,-176.321,9.155,148.782
C09838=1154.382,359.386,-80.507,-176.322,9.151,148.782
C09839=1154.386,359.138,-80.472,-176.325,9.147,148.781
C09840=1154.391,358.891,-80.437,-176.328,9.143,148.781
C09841=1154.394,358.643,-80.402,-176.330,9.139,148.781
C09842=1154.398,358.397,-80.367,-176.333,9.135,148.780
C09843=1154.402,358.149,-80.332,-176.335,9.132,148.780
C09844=1154.407,357.901,-80.298,-176.338,9.127,148.780
C09845=1154.410,357.654,-80.262,-176.340,9.124,148.780
C09846=1154.414,357.406,-80.228,-176.343,9.120,148.779
C09847=1154.418,357.158,-80.194,-176.345,9.116,148.779
C09848=1154.422,356.910,-80.159,-176.348,9.112,148.779
C09849=1154.426,356.664,-80.124,-176.351,9.108,148.778
C09850=1154.430,356.416,-80.089,-176.353,9.105,148.778
C09851=1154.434,356.168,-80.055,-176.355,9.101,148.778
C09852=1154.438,355.920,-80.020,-176.358,9.097,148.777
C09853=1154.442,355.673,-79.986,-176.360,9.093,148.777
C09854=1154.446,355.426,-79.951,-176.363,9.090,148.777
C09855=1154.450,355.178,-79.916,-176.365,9.086,148.776
C09856=1154.453,354.930,-79.882,-176.367,9.082,148.776
C09857=1154.458,354.683,-79.848,-176.370,9.078,148.776
C09858=1154.461,354.435,-79.813,-176.373,9.075,148.776
C09859=1154.466,354.188,-79.779,-176.375,9.070,148.775
C09860=1154.470,353.940,-79.744,-176.377,9.067,148.775
C09861=1154.474,353.692,-79.710,-176.380,9.063,148.775
C09862=1154.478,353.444,-79.675,-176.383,9.059,148.774
C09863=1154.482,353.197,-79.641,-176.385,9.055,148.774
C09864=1154.485,352.949,-79.607,-176.388,9.051,148.774
C09865=1154.490,352.702,-79.571,-176.390,9.048,148.774
C09866=1154.494,352.455,-79.538,-176.393,9.044,148.773
C09867=1154.498,352.206,-79.503,-176.395,9.040,148.773
C09868=1154.502,351.959,-79.470,-176.398,9.036,148.773
C09869=1154.505,351.711,-79.435,-176.400,9.033,148.772
C09870=1154.509,351.464,-79.401,-176.403,9.029,148.772
C09871=1154.513,351.216,-79.366,-176.405,9.025,148.772
C09872=1154.517,350.969,-79.332,-176.408,9.021,148.771
C09873=1154.522,350.721,-79.298,-176.410,9.018,148.771
C09874=1154.525,350.474,-79.263,-176.413,9.014,148.771
C09875=1154.529,350.226,-79.229,-176.415,9.010,148.771
C09876=1154.533,349.978,-79.195,-176.417,9.007,148.770
C09877=1154.538,349.730,-79.161,-176.420,9.003,148.770
C09878=1154.541,349.483,-79.127,-176.423,8.999,148.770
C09879=1154.545,349.235,-79.092,-176.425,8.995,148.770
C09880=1154.549,348.988,-79.058,-176.427,8.992,148.769
C09881=1154.554,348.741,-79.024,-176.430,8.987,148.769
C09882=1154.557,348.492,-78.990,-176.433,8.984,148.769
C09883=1154.562,348.245,-78.956,-176.435,8.980,148.768
C09884=1154.566,347.998,-78.922,-176.438,8.977,148.768
C09885=1154.569,347.750,-78.888,-176.440,8.972,148.768
C09886=1154.574,347.502,-78.854,-176.442,8.969,148.768
C09887=1154.578,347.255,-78.820,-176.445,8.965,148.767
C09888=1154.582,347.007,-78.785,-176.448,8.962,148.767
C09889=1154.586,346.759,-78.752,-176.451,8.958,148.767
C09890=1154.590,346.512,-78.718,-176.452,8.954,148.766
C09891=1154.594,346.264,-78.684,-176.455,8.950,148.766
C09892=1154.598,346.016,-78.650,-176.458,8.947,148.766
C09893=1154.602,345.769,-78.617,-176.460,8.943,148.766
C09894=1154.606,345.521,-78.583,-176.463,8.939,148.766
C09895=1154.610,345.273,-78.549,-176.465,8.936,148.765
C09896=1154.613,345.026,-78.515,-176.468,8.932,148.765
C09897=1154.618,344.778,-78.481,-176.470,8.928,148.765
C09898=1154.622,344.530,-78.447,-176.473,8.924,148.764
C09899=1154.626,344.282,-78.414,-176.475,8.921,148.764
C09900=1154.630,344.035,-78.380,-176.478,8.917,148.764
C09901=1154.634,343.787,-78.346,-176.480,8.914,148.764
C09902=1154.638,343.539,-78.312,-176.483,8.910,148.764
C09903=1154.642,343.292,-78.278,-176.485,8.906,148.763
C09904=1154.646,343.044,-78.245,-176.487,8.903,148.763
C09905=1154.651,342.796,-78.211,-176.490,8.899,148.763
C09906=1154.655,342.549,-78.178,-176.493,8.895,148.762
C09907=1154.658,342.301,-78.143,-176.496,8.891,148.762
C09908=1154.662,342.053,-78.110,-176.498,8.888,148.762
C09909=1154.667,341.805,-78.077,-176.500,8.885,148.762
C09910=1154.671,341.558,-78.043,-176.503,8.881,148.762
C09911=1154.675,341.310,-78.010,-176.505,8.877,148.761
C09912=1154.678,341.062,-77.976,-176.508,8.873,148.761
C09913=1154.682,340.815,-77.942,-176.510,8.870,148.761
C09914=1154.686,340.567,-77.909,-176.513,8.865,148.760
C09915=1154.691,340.319,-77.875,-176.515,8.862,148.760
C09916=1154.695,340.072,-77.841,-176.518,8.859,148.760
C09917=1154.699,339.792,-77.803,-176.521,8.855,148.760
C09918=1154.704,339.512,-77.766,-176.524,8.851,148.760
C09919=1154.709,339.231,-77.729,-176.526,8.847,148.759
C09920=1154.713,338.951,-77.691,-176.529,8.843,148.759
C09921=1154.717,338.704,-77.657,-176.532,8.838,148.759
C09922=1154.721,338.456,-77.624,-176.535,8.835,148.759
C09923=1154.725,338.209,-77.590,-176.537,8.832,148.758
C09924=1154.730,337.961,-77.557,-176.540,8.828,148.758
C09925=1154.734,337.713,-77.524,-176.542,8.824,148.758
C09926=1154.737,337.465,-77.491,-176.544,8.820,148.757
C09927=1154.741,337.217,-77.457,-176.547,8.817,148.757
C09928=1154.745,336.970,-77.424,-176.549,8.814,148.757
C09929=1154.749,336.722,-77.390,-176.552,8.809,148.757
C09930=1154.753,336.474,-77.357,-176.554,8.806,148.757
C09931=1154.758,336.227,-77.324,-176.557,8.802,148.756
C09932=1154.762,335.979,-77.291,-176.560,8.799,148.756
C09933=1154.766,335.731,-77.258,-176.562,8.795,148.756
C09934=1154.770,335.483,-77.225,-176.565,8.791,148.756
C09935=1154.774,335.236,-77.192,-176.567,8.788,148.756
C09936=1154.778,334.988,-77.158,-176.570,8.784,148.755
C09937=1154.782,334.740,-77.125,-176.572,8.781,148.755
C09938=1154.786,334.492,-77.092,-176.575,8.777,148.755
C09939=1154.790,334.244,-77.059,-176.577,8.773,148.755
C09940=1154.794,333.996,-77.025,-176.580,8.770,148.754
C09941=1154.798,333.748,-76.994,-176.582,8.767,148.754
C09942=1154.802,333.501,-76.960,-176.585,8.763,148.754
C09943=1154.806,333.253,-76.927,-176.587,8.759,148.754
C09944=1154.810,333.005,-76.894,-176.590,8.756,148.754
C09945=1154.815,332.757,-76.861,-176.593,8.752,148.753
C09946=1154.819,332.510,-76.828,-176.595,8.749,148.753
C09947=1154.823,332.262,-76.795,-176.598,8.745,148.753
C09948=1154.827,332.014,-76.763,-176.600,8.741,148.753
C09949=1154.831,331.766,-76.730,-176.602,8.738,148.752
C09950=1154.835,331.518,-76.696,-176.605,8.734,148.752
C09951=1154.839,331.271,-76.663,-176.608,8.731,148.752
C09952=1154.843,331.022,-76.631,-176.610,8.728,148.752
C09953=1154.847,330.775,-76.598,-176.613,8.724,148.752
C09954=1154.851,330.527,-76.565,-176.616,8.720,148.752
C09955=1154.856,330.280,-76.532,-176.618,8.717,148.751
C09956=1154.860,330.032,-76.500,-176.621,8.713,148.751
C09957=1154.864,329.784,-76.467,-176.623,8.710,148.751
C09958=1154.868,329.537,-76.434,-176.625,8.706,148.751
C09959=1154.872,329.288,-76.402,-176.628,8.702,148.751
C09960=1154.876,329.041,-76.369,-176.631,8.699,148.750
C09961=1154.880,328.793,-76.335,-176.633,8.696,148.750
C09962=1154.884,328.545,-76.304,-176.636,8.692,148.750
C09963=1154.888,328.297,-76.270,-176.638,8.688,148.750
C09964=1154.893,328.049,-76.238,-176.640,8.685,148.750
C09965=1154.896,327.801,-76.205,-176.644,8.681,148.749
C09966=1154.900,327.553,-76.173,-176.646,8.678,148.749
C09967=1154.905,327.305,-76.140,-176.648,8.675,148.749
C09968=1154.909,327.059,-76.108,-176.651,8.671,148.749
C09969=1154.913,326.810,-76.075,-176.654,8.667,148.749
C09970=1154.917,326.563,-76.042,-176.656,8.664,148.748
C09971=1154.921,326.314,-76.010,-176.659,8.660,148.748
C09972=1154.925,326.066,-75.978,-176.661,8.657,148.748
C09973=1154.929,325.819,-75.945,-176.663,8.654,148.748
C09974=1154.933,325.570,-75.913,-176.667,8.650,148.748
C09975=1154.938,325.323,-75.880,-176.669,8.646,148.748
C09976=1154.942,325.075,-75.848,-176.671,8.643,148.747
C09977=1154.946,324.828,-75.815,-176.674,8.639,148.747
C09978=1154.949,324.580,-75.783,-176.677,8.636,148.747
C09979=1154.954,324.331,-75.751,-176.679,8.633,148.747
C09980=1154.957,324.084,-75.718,-176.681,8.629,148.747
C09981=1154.962,323.836,-75.686,-176.685,8.625,148.747
C09982=1154.966,323.588,-75.654,-176.687,8.622,148.746
C09983=1154.970,323.340,-75.621,-176.689,8.619,148.746
C09984=1154.974,323.092,-75.589,-176.692,8.615,148.746
C09985=1154.978,322.844,-75.557,-176.694,8.612,148.746
C09986=1154.982,322.597,-75.524,-176.697,8.608,148.746
C09987=1154.987,322.349,-75.492,-176.700,8.604,148.745
C09988=1154.991,322.101,-75.460,-176.702,8.601,148.745
C09989=1154.995,321.852,-75.428,-176.705,8.598,148.745
C09990=1154.998,321.605,-75.395,-176.707,8.595,148.745
C09991=1155.003,321.357,-75.363,-176.710,8.591,148.745
C09992=1155.007,321.109,-75.331,-176.712,8.587,148.745
C09993=1155.012,320.861,-75.299,-176.715,8.584,148.745
C09994=1155.015,320.613,-75.267,-176.718,8.580,148.744
C09995=1155.020,320.366,-75.236,-176.720,8.577,148.744
C09996=1155.024,320.118,-75.202,-176.722,8.574,148.744
//INST
///DATE 2021/06/15 17:26
///ATTR SC,RW,RJ
////FRAME ROBOT
///GROUP1 RB1
NOP
MOVL C00000 V=800.0 PL=0
MOVL C00001 V=800.0 PL=0
MOVL C00002 V=800.0 PL=0
MOVL C00003 V=800.0 PL=0
MOVL C00004 V=800.0 PL=0
MOVL C00005 V=800.0 PL=0
MOVL C00006 V=800.0 PL=0
MOVL C00007 V=800.0 PL=0
MOVL C00008 V=800.0 PL=0
MOVL C00009 V=800.0 PL=0
MOVL C00010 V=800.0 PL=0
MOVL C00011 V=800.0 PL=0
MOVL C00012 V=800.0 PL=0
MOVL C00013 V=800.0 PL=0
MOVL C00014 V=800.0 PL=0
MOVL C00015 V=800.0 PL=0
MOVL C00016 V=800.0 PL=0
MOVL C00017 V=800.0 PL=0
MOVL C00018 V=800.0 PL=0
MOVL C00019 V=800.0 PL=0
MOVL C00020 V=800.0 PL=0
MOVL C00021 V=800.0 PL=0
MOVL C00022 V=800.0 PL=0
MOVL C00023 V=800.0 PL=0
MOVL C00024 V=800.0 PL=0
MOVL C00025 V=800.0 PL=0
MOVL C00026 V=800.0 PL=0
MOVL C00027 V=800.0 PL=0
MOVL C00028 V=800.0 PL=0
MOVL C00029 V=800.0 PL=0
MOVL C00030 V=800.0 PL=0
MOVL C00031 V=800.0 PL=0
MOVL C00032 V=800.0 PL=0
MOVL C00033 V=800.0 PL=0
MOVL C00034 V=800.0 PL=0
MOVL C00035 V=800.0 PL=0
MOVL C00036 V=800.0 PL=0
MOVL C00037 V=800.0 PL=0
MOVL C00038 V=800.0 PL=0
MOVL C00039 V=800.0 PL=0
MOVL C00040 V=800.0 PL=0
MOVL C00041 V=800.0 PL=0
MOVL C00042 V=800.0 PL=0
MOVL C00043 V=800.0 PL=0
MOVL C00044 V=800.0 PL=0
MOVL C00045 V=800.0 PL=0
MOVL C00046 V=800.0 PL=0
MOVL C00047 V=800.0 PL=0
MOVL C00048 V=800.0 PL=0
MOVL C00049 V=800.0 PL=0
MOVL C00050 V=800.0 PL=0
MOVL C00051 V=800.0 PL=0
MOVL C00052 V=800.0 PL=0
MOVL C00053 V=800.0 PL=0
MOVL C00054 V=800.0 PL=0
MOVL C00055 V=800.0 PL=0
MOVL C00056 V=800.0 PL=0
MOVL C00057 V=800.0 PL=0
MOVL C00058 V=800.0 PL=0
MOVL C00059 V=800.0 PL=0
MOVL C00060 V=800.0 PL=0
MOVL C00061 V=800.0 PL=0
MOVL C00062 V=800.0 PL=0
MOVL C00063 V=800.0 PL=0
MOVL C00064 V=800.0 PL=0
MOVL C00065 V=800.0 PL=0
MOVL C00066 V=800.0 PL=0
MOVL C00067 V=800.0 PL=0
MOVL C00068 V=800.0 PL=0
MOVL C00069 V=800.0 PL=0
MOVL C00070 V=800.0 PL=0
MOVL C00071 V=800.0 PL=0
MOVL C00072 V=800.0 PL=0
MOVL C00073 V=800.0 PL=0
MOVL C00074 V=800.0 PL=0
MOVL C00075 V=800.0 PL=0
MOVL C00076 V=800.0 PL=0
MOVL C00077 V=800.0 PL=0
MOVL C00078 V=800.0 PL=0
MOVL C00079 V=800.0 PL=0
MOVL C00080 V=800.0 PL=0
MOVL C00081 V=800.0 PL=0
MOVL C00082 V=800.0 PL=0
MOVL C00083 V=800.0 PL=0
MOVL C00084 V=800.0 PL=0
MOVL C00085 V=800.0 PL=0
MOVL C00086 V=800.0 PL=0
MOVL C00087 V=800.0 PL=0
MOVL C00088 V=800.0 PL=0
MOVL C00089 V=800.0 PL=0
MOVL C00090 V=800.0 PL=0
MOVL C00091 V=800.0 PL=0
MOVL C00092 V=800.0 PL=0
MOVL C00093 V=800.0 PL=0
MOVL C00094 V=800.0 PL=0
MOVL C00095 V=800.0 PL=0
MOVL C00096 V=800.0 PL=0
MOVL C00097 V=800.0 PL=0
MOVL C00098 V=800.0 PL=0
MOVL C00099 V=800.0 PL=0
MOVL C00100 V=800.0 PL=0
MOVL C00101 V=800.0 PL=0
MOVL C00102 V=800.0 PL=0
MOVL C00103 V=800.0 PL=0
MOVL C00104 V=800.0 PL=0
MOVL C00105 V=800.0 PL=0
MOVL C00106 V=800.0 PL=0
MOVL C00107 V=800.0 PL=0
MOVL C00108 V=800.0 PL=0
MOVL C00109 V=800.0 PL=0
MOVL C00110 V=800.0 PL=0
MOVL C00111 V=800.0 PL=0
MOVL C00112 V=800.0 PL=0
MOVL C00113 V=800.0 PL=0
MOVL C00114 V=800.0 PL=0
MOVL C00115 V=800.0 PL=0
MOVL C00116 V=800.0 PL=0
MOVL C00117 V=800.0 PL=0
MOVL C00118 V=800.0 PL=0
MOVL C00119 V=800.0 PL=0
MOVL C00120 V=800.0 PL=0
MOVL C00121 V=800.0 PL=0
MOVL C00122 V=800.0 PL=0
MOVL C00123 V=800.0 PL=0
MOVL C00124 V=800.0 PL=0
MOVL C00125 V=800.0 PL=0
MOVL C00126 V=800.0 PL=0
MOVL C00127 V=800.0 PL=0
MOVL C00128 V=800.0 PL=0
MOVL C00129 V=800.0 PL=0
MOVL C00130 V=800.0 PL=0
MOVL C00131 V=800.0 PL=0
MOVL C00132 V=800.0 PL=0
MOVL C00133 V=800.0 PL=0
MOVL C00134 V=800.0 PL=0
MOVL C00135 V=800.0 PL=0
MOVL C00136 V=800.0 PL=0
MOVL C00137 V=800.0 PL=0
MOVL C00138 V=800.0 PL=0
MOVL C00139 V=800.0 PL=0
MOVL C00140 V=800.0 PL=0
MOVL C00141 V=800.0 PL=0
MOVL C00142 V=800.0 PL=0
MOVL C00143 V=800.0 PL=0
MOVL C00144 V=800.0 PL=0
MOVL C00145 V=800.0 PL=0
MOVL C00146 V=800.0 PL=0
MOVL C00147 V=800.0 PL=0
MOVL C00148 V=800.0 PL=0
MOVL C00149 V=800.0 PL=0
MOVL C00150 V=800.0 PL=0
MOVL C00151 V=800.0 PL=0
MOVL C00152 V=800.0 PL=0
MOVL C00153 V=800.0 PL=0
MOVL C00154 V=800.0 PL=0
MOVL C00155 V=800.0 PL=0
MOVL C00156 V=800.0 PL=0
MOVL C00157 V=800.0 PL=0
MOVL C00158 V=800.0 PL=0
MOVL C00159 V=800.0 PL=0
MOVL C00160 V=800.0 PL=0
MOVL C00161 V=800.0 PL=0
MOVL C00162 V=800.0 PL=0
MOVL C00163 V=800.0 PL=0
MOVL C00164 V=800.0 PL=0
MOVL C00165 V=800.0 PL=0
MOVL C00166 V=800.0 PL=0
MOVL C00167 V=800.0 PL=0
MOVL C00168 V=800.0 PL=0
MOVL C00169 V=800.0 PL=0
MOVL C00170 V=800.0 PL=0
MOVL C00171 V=800.0 PL=0
MOVL C00172 V=800.0 PL=0
MOVL C00173 V=800.0 PL=0
MOVL C00174 V=800.0 PL=0
MOVL C00175 V=800.0 PL=0
MOVL C00176 V=800.0 PL=0
MOVL C00177 V=800.0 PL=0
MOVL C00178 V=800.0 PL=0
MOVL C00179 V=800.0 PL=0
MOVL C00180 V=800.0 PL=0
MOVL C00181 V=800.0 PL=0
MOVL C00182 V=800.0 PL=0
MOVL C00183 V=800.0 PL=0
MOVL C00184 V=800.0 PL=0
MOVL C00185 V=800.0 PL=0
MOVL C00186 V=800.0 PL=0
MOVL C00187 V=800.0 PL=0
MOVL C00188 V=800.0 PL=0
MOVL C00189 V=800.0 PL=0
MOVL C00190 V=800.0 PL=0
MOVL C00191 V=800.0 PL=0
MOVL C00192 V=800.0 PL=0
MOVL C00193 V=800.0 PL=0
MOVL C00194 V=800.0 PL=0
MOVL C00195 V=800.0 PL=0
MOVL C00196 V=800.0 PL=0
MOVL C00197 V=800.0 PL=0
MOVL C00198 V=800.0 PL=0
MOVL C00199 V=800.0 PL=0
MOVL C00200 V=800.0 PL=0
MOVL C00201 V=800.0 PL=0
MOVL C00202 V=800.0 PL=0
MOVL C00203 V=800.0 PL=0
MOVL C00204 V=800.0 PL=0
MOVL C00205 V=800.0 PL=0
MOVL C00206 V=800.0 PL=0
MOVL C00207 V=800.0 PL=0
MOVL C00208 V=800.0 PL=0
MOVL C00209 V=800.0 PL=0
MOVL C00210 V=800.0 PL=0
MOVL C00211 V=800.0 PL=0
MOVL C00212 V=800.0 PL=0
MOVL C00213 V=800.0 PL=0
MOVL C00214 V=800.0 PL=0
MOVL C00215 V=800.0 PL=0
MOVL C00216 V=800.0 PL=0
MOVL C00217 V=800.0 PL=0
MOVL C00218 V=800.0 PL=0
MOVL C00219 V=800.0 PL=0
MOVL C00220 V=800.0 PL=0
MOVL C00221 V=800.0 PL=0
MOVL C00222 V=800.0 PL=0
MOVL C00223 V=800.0 PL=0
MOVL C00224 V=800.0 PL=0
MOVL C00225 V=800.0 PL=0
MOVL C00226 V=800.0 PL=0
MOVL C00227 V=800.0 PL=0
MOVL C00228 V=800.0 PL=0
MOVL C00229 V=800.0 PL=0
MOVL C00230 V=800.0 PL=0
MOVL C00231 V=800.0 PL=0
MOVL C00232 V=800.0 PL=0
MOVL C00233 V=800.0 PL=0
MOVL C00234 V=800.0 PL=0
MOVL C00235 V=800.0 PL=0
MOVL C00236 V=800.0 PL=0
MOVL C00237 V=800.0 PL=0
MOVL C00238 V=800.0 PL=0
MOVL C00239 V=800.0 PL=0
MOVL C00240 V=800.0 PL=0
MOVL C00241 V=800.0 PL=0
MOVL C00242 V=800.0 PL=0
MOVL C00243 V=800.0 PL=0
MOVL C00244 V=800.0 PL=0
MOVL C00245 V=800.0 PL=0
MOVL C00246 V=800.0 PL=0
MOVL C00247 V=800.0 PL=0
MOVL C00248 V=800.0 PL=0
MOVL C00249 V=800.0 PL=0
MOVL C00250 V=800.0 PL=0
MOVL C00251 V=800.0 PL=0
MOVL C00252 V=800.0 PL=0
MOVL C00253 V=800.0 PL=0
MOVL C00254 V=800.0 PL=0
MOVL C00255 V=800.0 PL=0
MOVL C00256 V=800.0 PL=0
MOVL C00257 V=800.0 PL=0
MOVL C00258 V=800.0 PL=0
MOVL C00259 V=800.0 PL=0
MOVL C00260 V=800.0 PL=0
MOVL C00261 V=800.0 PL=0
MOVL C00262 V=800.0 PL=0
MOVL C00263 V=800.0 PL=0
MOVL C00264 V=800.0 PL=0
MOVL C00265 V=800.0 PL=0
MOVL C00266 V=800.0 PL=0
MOVL C00267 V=800.0 PL=0
MOVL C00268 V=800.0 PL=0
MOVL C00269 V=800.0 PL=0
MOVL C00270 V=800.0 PL=0
MOVL C00271 V=800.0 PL=0
MOVL C00272 V=800.0 PL=0
MOVL C00273 V=800.0 PL=0
MOVL C00274 V=800.0 PL=0
MOVL C00275 V=800.0 PL=0
MOVL C00276 V=800.0 PL=0
MOVL C00277 V=800.0 PL=0
MOVL C00278 V=800.0 PL=0
MOVL C00279 V=800.0 PL=0
MOVL C00280 V=800.0 PL=0
MOVL C00281 V=800.0 PL=0
MOVL C00282 V=800.0 PL=0
MOVL C00283 V=800.0 PL=0
MOVL C00284 V=800.0 PL=0
MOVL C00285 V=800.0 PL=0
MOVL C00286 V=800.0 PL=0
MOVL C00287 V=800.0 PL=0
MOVL C00288 V=800.0 PL=0
MOVL C00289 V=800.0 PL=0
MOVL C00290 V=800.0 PL=0
MOVL C00291 V=800.0 PL=0
MOVL C00292 V=800.0 PL=0
MOVL C00293 V=800.0 PL=0
MOVL C00294 V=800.0 PL=0
MOVL C00295 V=800.0 PL=0
MOVL C00296 V=800.0 PL=0
MOVL C00297 V=800.0 PL=0
MOVL C00298 V=800.0 PL=0
MOVL C00299 V=800.0 PL=0
MOVL C00300 V=800.0 PL=0
MOVL C00301 V=800.0 PL=0
MOVL C00302 V=800.0 PL=0
MOVL C00303 V=800.0 PL=0
MOVL C00304 V=800.0 PL=0
MOVL C00305 V=800.0 PL=0
MOVL C00306 V=800.0 PL=0
MOVL C00307 V=800.0 PL=0
MOVL C00308 V=800.0 PL=0
MOVL C00309 V=800.0 PL=0
MOVL C00310 V=800.0 PL=0
MOVL C00311 V=800.0 PL=0
MOVL C00312 V=800.0 PL=0
MOVL C00313 V=800.0 PL=0
MOVL C00314 V=800.0 PL=0
MOVL C00315 V=800.0 PL=0
MOVL C00316 V=800.0 PL=0
MOVL C00317 V=800.0 PL=0
MOVL C00318 V=800.0 PL=0
MOVL C00319 V=800.0 PL=0
MOVL C00320 V=800.0 PL=0
MOVL C00321 V=800.0 PL=0
MOVL C00322 V=800.0 PL=0
MOVL C00323 V=800.0 PL=0
MOVL C00324 V=800.0 PL=0
MOVL C00325 V=800.0 PL=0
MOVL C00326 V=800.0 PL=0
MOVL C00327 V=800.0 PL=0
MOVL C00328 V=800.0 PL=0
MOVL C00329 V=800.0 PL=0
MOVL C00330 V=800.0 PL=0
MOVL C00331 V=800.0 PL=0
MOVL C00332 V=800.0 PL=0
MOVL C00333 V=800.0 PL=0
MOVL C00334 V=800.0 PL=0
MOVL C00335 V=800.0 PL=0
MOVL C00336 V=800.0 PL=0
MOVL C00337 V=800.0 PL=0
MOVL C00338 V=800.0 PL=0
MOVL C00339 V=800.0 PL=0
MOVL C00340 V=800.0 PL=0
MOVL C00341 V=800.0 PL=0
MOVL C00342 V=800.0 PL=0
MOVL C00343 V=800.0 PL=0
MOVL C00344 V=800.0 PL=0
MOVL C00345 V=800.0 PL=0
MOVL C00346 V=800.0 PL=0
MOVL C00347 V=800.0 PL=0
MOVL C00348 V=800.0 PL=0
MOVL C00349 V=800.0 PL=0
MOVL C00350 V=800.0 PL=0
MOVL C00351 V=800.0 PL=0
MOVL C00352 V=800.0 PL=0
MOVL C00353 V=800.0 PL=0
MOVL C00354 V=800.0 PL=0
MOVL C00355 V=800.0 PL=0
MOVL C00356 V=800.0 PL=0
MOVL C00357 V=800.0 PL=0
MOVL C00358 V=800.0 PL=0
MOVL C00359 V=800.0 PL=0
MOVL C00360 V=800.0 PL=0
MOVL C00361 V=800.0 PL=0
MOVL C00362 V=800.0 PL=0
MOVL C00363 V=800.0 PL=0
MOVL C00364 V=800.0 PL=0
MOVL C00365 V=800.0 PL=0
MOVL C00366 V=800.0 PL=0
MOVL C00367 V=800.0 PL=0
MOVL C00368 V=800.0 PL=0
MOVL C00369 V=800.0 PL=0
MOVL C00370 V=800.0 PL=0
MOVL C00371 V=800.0 PL=0
MOVL C00372 V=800.0 PL=0
MOVL C00373 V=800.0 PL=0
MOVL C00374 V=800.0 PL=0
MOVL C00375 V=800.0 PL=0
MOVL C00376 V=800.0 PL=0
MOVL C00377 V=800.0 PL=0
MOVL C00378 V=800.0 PL=0
MOVL C00379 V=800.0 PL=0
MOVL C00380 V=800.0 PL=0
MOVL C00381 V=800.0 PL=0
MOVL C00382 V=800.0 PL=0
MOVL C00383 V=800.0 PL=0
MOVL C00384 V=800.0 PL=0
MOVL C00385 V=800.0 PL=0
MOVL C00386 V=800.0 PL=0
MOVL C00387 V=800.0 PL=0
MOVL C00388 V=800.0 PL=0
MOVL C00389 V=800.0 PL=0
MOVL C00390 V=800.0 PL=0
MOVL C00391 V=800.0 PL=0
MOVL C00392 V=800.0 PL=0
MOVL C00393 V=800.0 PL=0
MOVL C00394 V=800.0 PL=0
MOVL C00395 V=800.0 PL=0
MOVL C00396 V=800.0 PL=0
MOVL C00397 V=800.0 PL=0
MOVL C00398 V=800.0 PL=0
MOVL C00399 V=800.0 PL=0
MOVL C00400 V=800.0 PL=0
MOVL C00401 V=800.0 PL=0
MOVL C00402 V=800.0 PL=0
MOVL C00403 V=800.0 PL=0
MOVL C00404 V=800.0 PL=0
MOVL C00405 V=800.0 PL=0
MOVL C00406 V=800.0 PL=0
MOVL C00407 V=800.0 PL=0
MOVL C00408 V=800.0 PL=0
MOVL C00409 V=800.0 PL=0
MOVL C00410 V=800.0 PL=0
MOVL C00411 V=800.0 PL=0
MOVL C00412 V=800.0 PL=0
MOVL C00413 V=800.0 PL=0
MOVL C00414 V=800.0 PL=0
MOVL C00415 V=800.0 PL=0
MOVL C00416 V=800.0 PL=0
MOVL C00417 V=800.0 PL=0
MOVL C00418 V=800.0 PL=0
MOVL C00419 V=800.0 PL=0
MOVL C00420 V=800.0 PL=0
MOVL C00421 V=800.0 PL=0
MOVL C00422 V=800.0 PL=0
MOVL C00423 V=800.0 PL=0
MOVL C00424 V=800.0 PL=0
MOVL C00425 V=800.0 PL=0
MOVL C00426 V=800.0 PL=0
MOVL C00427 V=800.0 PL=0
MOVL C00428 V=800.0 PL=0
MOVL C00429 V=800.0 PL=0
MOVL C00430 V=800.0 PL=0
MOVL C00431 V=800.0 PL=0
MOVL C00432 V=800.0 PL=0
MOVL C00433 V=800.0 PL=0
MOVL C00434 V=800.0 PL=0
MOVL C00435 V=800.0 PL=0
MOVL C00436 V=800.0 PL=0
MOVL C00437 V=800.0 PL=0
MOVL C00438 V=800.0 PL=0
MOVL C00439 V=800.0 PL=0
MOVL C00440 V=800.0 PL=0
MOVL C00441 V=800.0 PL=0
MOVL C00442 V=800.0 PL=0
MOVL C00443 V=800.0 PL=0
MOVL C00444 V=800.0 PL=0
MOVL C00445 V=800.0 PL=0
MOVL C00446 V=800.0 PL=0
MOVL C00447 V=800.0 PL=0
MOVL C00448 V=800.0 PL=0
MOVL C00449 V=800.0 PL=0
MOVL C00450 V=800.0 PL=0
MOVL C00451 V=800.0 PL=0
MOVL C00452 V=800.0 PL=0
MOVL C00453 V=800.0 PL=0
MOVL C00454 V=800.0 PL=0
MOVL C00455 V=800.0 PL=0
MOVL C00456 V=800.0 PL=0
MOVL C00457 V=800.0 PL=0
MOVL C00458 V=800.0 PL=0
MOVL C00459 V=800.0 PL=0
MOVL C00460 V=800.0 PL=0
MOVL C00461 V=800.0 PL=0
MOVL C00462 V=800.0 PL=0
MOVL C00463 V=800.0 PL=0
MOVL C00464 V=800.0 PL=0
MOVL C00465 V=800.0 PL=0
MOVL C00466 V=800.0 PL=0
MOVL C00467 V=800.0 PL=0
MOVL C00468 V=800.0 PL=0
MOVL C00469 V=800.0 PL=0
MOVL C00470 V=800.0 PL=0
MOVL C00471 V=800.0 PL=0
MOVL C00472 V=800.0 PL=0
MOVL C00473 V=800.0 PL=0
MOVL C00474 V=800.0 PL=0
MOVL C00475 V=800.0 PL=0
MOVL C00476 V=800.0 PL=0
MOVL C00477 V=800.0 PL=0
MOVL C00478 V=800.0 PL=0
MOVL C00479 V=800.0 PL=0
MOVL C00480 V=800.0 PL=0
MOVL C00481 V=800.0 PL=0
MOVL C00482 V=800.0 PL=0
MOVL C00483 V=800.0 PL=0
MOVL C00484 V=800.0 PL=0
MOVL C00485 V=800.0 PL=0
MOVL C00486 V=800.0 PL=0
MOVL C00487 V=800.0 PL=0
MOVL C00488 V=800.0 PL=0
MOVL C00489 V=800.0 PL=0
MOVL C00490 V=800.0 PL=0
MOVL C00491 V=800.0 PL=0
MOVL C00492 V=800.0 PL=0
MOVL C00493 V=800.0 PL=0
MOVL C00494 V=800.0 PL=0
MOVL C00495 V=800.0 PL=0
MOVL C00496 V=800.0 PL=0
MOVL C00497 V=800.0 PL=0
MOVL C00498 V=800.0 PL=0
MOVL C00499 V=800.0 PL=0
MOVL C00500 V=800.0 PL=0
MOVL C00501 V=800.0 PL=0
MOVL C00502 V=800.0 PL=0
MOVL C00503 V=800.0 PL=0
MOVL C00504 V=800.0 PL=0
MOVL C00505 V=800.0 PL=0
MOVL C00506 V=800.0 PL=0
MOVL C00507 V=800.0 PL=0
MOVL C00508 V=800.0 PL=0
MOVL C00509 V=800.0 PL=0
MOVL C00510 V=800.0 PL=0
MOVL C00511 V=800.0 PL=0
MOVL C00512 V=800.0 PL=0
MOVL C00513 V=800.0 PL=0
MOVL C00514 V=800.0 PL=0
MOVL C00515 V=800.0 PL=0
MOVL C00516 V=800.0 PL=0
MOVL C00517 V=800.0 PL=0
MOVL C00518 V=800.0 PL=0
MOVL C00519 V=800.0 PL=0
MOVL C00520 V=800.0 PL=0
MOVL C00521 V=800.0 PL=0
MOVL C00522 V=800.0 PL=0
MOVL C00523 V=800.0 PL=0
MOVL C00524 V=800.0 PL=0
MOVL C00525 V=800.0 PL=0
MOVL C00526 V=800.0 PL=0
MOVL C00527 V=800.0 PL=0
MOVL C00528 V=800.0 PL=0
MOVL C00529 V=800.0 PL=0
MOVL C00530 V=800.0 PL=0
MOVL C00531 V=800.0 PL=0
MOVL C00532 V=800.0 PL=0
MOVL C00533 V=800.0 PL=0
MOVL C00534 V=800.0 PL=0
MOVL C00535 V=800.0 PL=0
MOVL C00536 V=800.0 PL=0
MOVL C00537 V=800.0 PL=0
MOVL C00538 V=800.0 PL=0
MOVL C00539 V=800.0 PL=0
MOVL C00540 V=800.0 PL=0
MOVL C00541 V=800.0 PL=0
MOVL C00542 V=800.0 PL=0
MOVL C00543 V=800.0 PL=0
MOVL C00544 V=800.0 PL=0
MOVL C00545 V=800.0 PL=0
MOVL C00546 V=800.0 PL=0
MOVL C00547 V=800.0 PL=0
MOVL C00548 V=800.0 PL=0
MOVL C00549 V=800.0 PL=0
MOVL C00550 V=800.0 PL=0
MOVL C00551 V=800.0 PL=0
MOVL C00552 V=800.0 PL=0
MOVL C00553 V=800.0 PL=0
MOVL C00554 V=800.0 PL=0
MOVL C00555 V=800.0 PL=0
MOVL C00556 V=800.0 PL=0
MOVL C00557 V=800.0 PL=0
MOVL C00558 V=800.0 PL=0
MOVL C00559 V=800.0 PL=0
MOVL C00560 V=800.0 PL=0
MOVL C00561 V=800.0 PL=0
MOVL C00562 V=800.0 PL=0
MOVL C00563 V=800.0 PL=0
MOVL C00564 V=800.0 PL=0
MOVL C00565 V=800.0 PL=0
MOVL C00566 V=800.0 PL=0
MOVL C00567 V=800.0 PL=0
MOVL C00568 V=800.0 PL=0
MOVL C00569 V=800.0 PL=0
MOVL C00570 V=800.0 PL=0
MOVL C00571 V=800.0 PL=0
MOVL C00572 V=800.0 PL=0
MOVL C00573 V=800.0 PL=0
MOVL C00574 V=800.0 PL=0
MOVL C00575 V=800.0 PL=0
MOVL C00576 V=800.0 PL=0
MOVL C00577 V=800.0 PL=0
MOVL C00578 V=800.0 PL=0
MOVL C00579 V=800.0 PL=0
MOVL C00580 V=800.0 PL=0
MOVL C00581 V=800.0 PL=0
MOVL C00582 V=800.0 PL=0
MOVL C00583 V=800.0 PL=0
MOVL C00584 V=800.0 PL=0
MOVL C00585 V=800.0 PL=0
MOVL C00586 V=800.0 PL=0
MOVL C00587 V=800.0 PL=0
MOVL C00588 V=800.0 PL=0
MOVL C00589 V=800.0 PL=0
MOVL C00590 V=800.0 PL=0
MOVL C00591 V=800.0 PL=0
MOVL C00592 V=800.0 PL=0
MOVL C00593 V=800.0 PL=0
MOVL C00594 V=800.0 PL=0
MOVL C00595 V=800.0 PL=0
MOVL C00596 V=800.0 PL=0
MOVL C00597 V=800.0 PL=0
MOVL C00598 V=800.0 PL=0
MOVL C00599 V=800.0 PL=0
MOVL C00600 V=800.0 PL=0
MOVL C00601 V=800.0 PL=0
MOVL C00602 V=800.0 PL=0
MOVL C00603 V=800.0 PL=0
MOVL C00604 V=800.0 PL=0
MOVL C00605 V=800.0 PL=0
MOVL C00606 V=800.0 PL=0
MOVL C00607 V=800.0 PL=0
MOVL C00608 V=800.0 PL=0
MOVL C00609 V=800.0 PL=0
MOVL C00610 V=800.0 PL=0
MOVL C00611 V=800.0 PL=0
MOVL C00612 V=800.0 PL=0
MOVL C00613 V=800.0 PL=0
MOVL C00614 V=800.0 PL=0
MOVL C00615 V=800.0 PL=0
MOVL C00616 V=800.0 PL=0
MOVL C00617 V=800.0 PL=0
MOVL C00618 V=800.0 PL=0
MOVL C00619 V=800.0 PL=0
MOVL C00620 V=800.0 PL=0
MOVL C00621 V=800.0 PL=0
MOVL C00622 V=800.0 PL=0
MOVL C00623 V=800.0 PL=0
MOVL C00624 V=800.0 PL=0
MOVL C00625 V=800.0 PL=0
MOVL C00626 V=800.0 PL=0
MOVL C00627 V=800.0 PL=0
MOVL C00628 V=800.0 PL=0
MOVL C00629 V=800.0 PL=0
MOVL C00630 V=800.0 PL=0
MOVL C00631 V=800.0 PL=0
MOVL C00632 V=800.0 PL=0
MOVL C00633 V=800.0 PL=0
MOVL C00634 V=800.0 PL=0
MOVL C00635 V=800.0 PL=0
MOVL C00636 V=800.0 PL=0
MOVL C00637 V=800.0 PL=0
MOVL C00638 V=800.0 PL=0
MOVL C00639 V=800.0 PL=0
MOVL C00640 V=800.0 PL=0
MOVL C00641 V=800.0 PL=0
MOVL C00642 V=800.0 PL=0
MOVL C00643 V=800.0 PL=0
MOVL C00644 V=800.0 PL=0
MOVL C00645 V=800.0 PL=0
MOVL C00646 V=800.0 PL=0
MOVL C00647 V=800.0 PL=0
MOVL C00648 V=800.0 PL=0
MOVL C00649 V=800.0 PL=0
MOVL C00650 V=800.0 PL=0
MOVL C00651 V=800.0 PL=0
MOVL C00652 V=800.0 PL=0
MOVL C00653 V=800.0 PL=0
MOVL C00654 V=800.0 PL=0
MOVL C00655 V=800.0 PL=0
MOVL C00656 V=800.0 PL=0
MOVL C00657 V=800.0 PL=0
MOVL C00658 V=800.0 PL=0
MOVL C00659 V=800.0 PL=0
MOVL C00660 V=800.0 PL=0
MOVL C00661 V=800.0 PL=0
MOVL C00662 V=800.0 PL=0
MOVL C00663 V=800.0 PL=0
MOVL C00664 V=800.0 PL=0
MOVL C00665 V=800.0 PL=0
MOVL C00666 V=800.0 PL=0
MOVL C00667 V=800.0 PL=0
MOVL C00668 V=800.0 PL=0
MOVL C00669 V=800.0 PL=0
MOVL C00670 V=800.0 PL=0
MOVL C00671 V=800.0 PL=0
MOVL C00672 V=800.0 PL=0
MOVL C00673 V=800.0 PL=0
MOVL C00674 V=800.0 PL=0
MOVL C00675 V=800.0 PL=0
MOVL C00676 V=800.0 PL=0
MOVL C00677 V=800.0 PL=0
MOVL C00678 V=800.0 PL=0
MOVL C00679 V=800.0 PL=0
MOVL C00680 V=800.0 PL=0
MOVL C00681 V=800.0 PL=0
MOVL C00682 V=800.0 PL=0
MOVL C00683 V=800.0 PL=0
MOVL C00684 V=800.0 PL=0
MOVL C00685 V=800.0 PL=0
MOVL C00686 V=800.0 PL=0
MOVL C00687 V=800.0 PL=0
MOVL C00688 V=800.0 PL=0
MOVL C00689 V=800.0 PL=0
MOVL C00690 V=800.0 PL=0
MOVL C00691 V=800.0 PL=0
MOVL C00692 V=800.0 PL=0
MOVL C00693 V=800.0 PL=0
MOVL C00694 V=800.0 PL=0
MOVL C00695 V=800.0 PL=0
MOVL C00696 V=800.0 PL=0
MOVL C00697 V=800.0 PL=0
MOVL C00698 V=800.0 PL=0
MOVL C00699 V=800.0 PL=0
MOVL C00700 V=800.0 PL=0
MOVL C00701 V=800.0 PL=0
MOVL C00702 V=800.0 PL=0
MOVL C00703 V=800.0 PL=0
MOVL C00704 V=800.0 PL=0
MOVL C00705 V=800.0 PL=0
MOVL C00706 V=800.0 PL=0
MOVL C00707 V=800.0 PL=0
MOVL C00708 V=800.0 PL=0
MOVL C00709 V=800.0 PL=0
MOVL C00710 V=800.0 PL=0
MOVL C00711 V=800.0 PL=0
MOVL C00712 V=800.0 PL=0
MOVL C00713 V=800.0 PL=0
MOVL C00714 V=800.0 PL=0
MOVL C00715 V=800.0 PL=0
MOVL C00716 V=800.0 PL=0
MOVL C00717 V=800.0 PL=0
MOVL C00718 V=800.0 PL=0
MOVL C00719 V=800.0 PL=0
MOVL C00720 V=800.0 PL=0
MOVL C00721 V=800.0 PL=0
MOVL C00722 V=800.0 PL=0
MOVL C00723 V=800.0 PL=0
MOVL C00724 V=800.0 PL=0
MOVL C00725 V=800.0 PL=0
MOVL C00726 V=800.0 PL=0
MOVL C00727 V=800.0 PL=0
MOVL C00728 V=800.0 PL=0
MOVL C00729 V=800.0 PL=0
MOVL C00730 V=800.0 PL=0
MOVL C00731 V=800.0 PL=0
MOVL C00732 V=800.0 PL=0
MOVL C00733 V=800.0 PL=0
MOVL C00734 V=800.0 PL=0
MOVL C00735 V=800.0 PL=0
MOVL C00736 V=800.0 PL=0
MOVL C00737 V=800.0 PL=0
MOVL C00738 V=800.0 PL=0
MOVL C00739 V=800.0 PL=0
MOVL C00740 V=800.0 PL=0
MOVL C00741 V=800.0 PL=0
MOVL C00742 V=800.0 PL=0
MOVL C00743 V=800.0 PL=0
MOVL C00744 V=800.0 PL=0
MOVL C00745 V=800.0 PL=0
MOVL C00746 V=800.0 PL=0
MOVL C00747 V=800.0 PL=0
MOVL C00748 V=800.0 PL=0
MOVL C00749 V=800.0 PL=0
MOVL C00750 V=800.0 PL=0
MOVL C00751 V=800.0 PL=0
MOVL C00752 V=800.0 PL=0
MOVL C00753 V=800.0 PL=0
MOVL C00754 V=800.0 PL=0
MOVL C00755 V=800.0 PL=0
MOVL C00756 V=800.0 PL=0
MOVL C00757 V=800.0 PL=0
MOVL C00758 V=800.0 PL=0
MOVL C00759 V=800.0 PL=0
MOVL C00760 V=800.0 PL=0
MOVL C00761 V=800.0 PL=0
MOVL C00762 V=800.0 PL=0
MOVL C00763 V=800.0 PL=0
MOVL C00764 V=800.0 PL=0
MOVL C00765 V=800.0 PL=0
MOVL C00766 V=800.0 PL=0
MOVL C00767 V=800.0 PL=0
MOVL C00768 V=800.0 PL=0
MOVL C00769 V=800.0 PL=0
MOVL C00770 V=800.0 PL=0
MOVL C00771 V=800.0 PL=0
MOVL C00772 V=800.0 PL=0
MOVL C00773 V=800.0 PL=0
MOVL C00774 V=800.0 PL=0
MOVL C00775 V=800.0 PL=0
MOVL C00776 V=800.0 PL=0
MOVL C00777 V=800.0 PL=0
MOVL C00778 V=800.0 PL=0
MOVL C00779 V=800.0 PL=0
MOVL C00780 V=800.0 PL=0
MOVL C00781 V=800.0 PL=0
MOVL C00782 V=800.0 PL=0
MOVL C00783 V=800.0 PL=0
MOVL C00784 V=800.0 PL=0
MOVL C00785 V=800.0 PL=0
MOVL C00786 V=800.0 PL=0
MOVL C00787 V=800.0 PL=0
MOVL C00788 V=800.0 PL=0
MOVL C00789 V=800.0 PL=0
MOVL C00790 V=800.0 PL=0
MOVL C00791 V=800.0 PL=0
MOVL C00792 V=800.0 PL=0
MOVL C00793 V=800.0 PL=0
MOVL C00794 V=800.0 PL=0
MOVL C00795 V=800.0 PL=0
MOVL C00796 V=800.0 PL=0
MOVL C00797 V=800.0 PL=0
MOVL C00798 V=800.0 PL=0
MOVL C00799 V=800.0 PL=0
MOVL C00800 V=800.0 PL=0
MOVL C00801 V=800.0 PL=0
MOVL C00802 V=800.0 PL=0
MOVL C00803 V=800.0 PL=0
MOVL C00804 V=800.0 PL=0
MOVL C00805 V=800.0 PL=0
MOVL C00806 V=800.0 PL=0
MOVL C00807 V=800.0 PL=0
MOVL C00808 V=800.0 PL=0
MOVL C00809 V=800.0 PL=0
MOVL C00810 V=800.0 PL=0
MOVL C00811 V=800.0 PL=0
MOVL C00812 V=800.0 PL=0
MOVL C00813 V=800.0 PL=0
MOVL C00814 V=800.0 PL=0
MOVL C00815 V=800.0 PL=0
MOVL C00816 V=800.0 PL=0
MOVL C00817 V=800.0 PL=0
MOVL C00818 V=800.0 PL=0
MOVL C00819 V=800.0 PL=0
MOVL C00820 V=800.0 PL=0
MOVL C00821 V=800.0 PL=0
MOVL C00822 V=800.0 PL=0
MOVL C00823 V=800.0 PL=0
MOVL C00824 V=800.0 PL=0
MOVL C00825 V=800.0 PL=0
MOVL C00826 V=800.0 PL=0
MOVL C00827 V=800.0 PL=0
MOVL C00828 V=800.0 PL=0
MOVL C00829 V=800.0 PL=0
MOVL C00830 V=800.0 PL=0
MOVL C00831 V=800.0 PL=0
MOVL C00832 V=800.0 PL=0
MOVL C00833 V=800.0 PL=0
MOVL C00834 V=800.0 PL=0
MOVL C00835 V=800.0 PL=0
MOVL C00836 V=800.0 PL=0
MOVL C00837 V=800.0 PL=0
MOVL C00838 V=800.0 PL=0
MOVL C00839 V=800.0 PL=0
MOVL C00840 V=800.0 PL=0
MOVL C00841 V=800.0 PL=0
MOVL C00842 V=800.0 PL=0
MOVL C00843 V=800.0 PL=0
MOVL C00844 V=800.0 PL=0
MOVL C00845 V=800.0 PL=0
MOVL C00846 V=800.0 PL=0
MOVL C00847 V=800.0 PL=0
MOVL C00848 V=800.0 PL=0
MOVL C00849 V=800.0 PL=0
MOVL C00850 V=800.0 PL=0
MOVL C00851 V=800.0 PL=0
MOVL C00852 V=800.0 PL=0
MOVL C00853 V=800.0 PL=0
MOVL C00854 V=800.0 PL=0
MOVL C00855 V=800.0 PL=0
MOVL C00856 V=800.0 PL=0
MOVL C00857 V=800.0 PL=0
MOVL C00858 V=800.0 PL=0
MOVL C00859 V=800.0 PL=0
MOVL C00860 V=800.0 PL=0
MOVL C00861 V=800.0 PL=0
MOVL C00862 V=800.0 PL=0
MOVL C00863 V=800.0 PL=0
MOVL C00864 V=800.0 PL=0
MOVL C00865 V=800.0 PL=0
MOVL C00866 V=800.0 PL=0
MOVL C00867 V=800.0 PL=0
MOVL C00868 V=800.0 PL=0
MOVL C00869 V=800.0 PL=0
MOVL C00870 V=800.0 PL=0
MOVL C00871 V=800.0 PL=0
MOVL C00872 V=800.0 PL=0
MOVL C00873 V=800.0 PL=0
MOVL C00874 V=800.0 PL=0
MOVL C00875 V=800.0 PL=0
MOVL C00876 V=800.0 PL=0
MOVL C00877 V=800.0 PL=0
MOVL C00878 V=800.0 PL=0
MOVL C00879 V=800.0 PL=0
MOVL C00880 V=800.0 PL=0
MOVL C00881 V=800.0 PL=0
MOVL C00882 V=800.0 PL=0
MOVL C00883 V=800.0 PL=0
MOVL C00884 V=800.0 PL=0
MOVL C00885 V=800.0 PL=0
MOVL C00886 V=800.0 PL=0
MOVL C00887 V=800.0 PL=0
MOVL C00888 V=800.0 PL=0
MOVL C00889 V=800.0 PL=0
MOVL C00890 V=800.0 PL=0
MOVL C00891 V=800.0 PL=0
MOVL C00892 V=800.0 PL=0
MOVL C00893 V=800.0 PL=0
MOVL C00894 V=800.0 PL=0
MOVL C00895 V=800.0 PL=0
MOVL C00896 V=800.0 PL=0
MOVL C00897 V=800.0 PL=0
MOVL C00898 V=800.0 PL=0
MOVL C00899 V=800.0 PL=0
MOVL C00900 V=800.0 PL=0
MOVL C00901 V=800.0 PL=0
MOVL C00902 V=800.0 PL=0
MOVL C00903 V=800.0 PL=0
MOVL C00904 V=800.0 PL=0
MOVL C00905 V=800.0 PL=0
MOVL C00906 V=800.0 PL=0
MOVL C00907 V=800.0 PL=0
MOVL C00908 V=800.0 PL=0
MOVL C00909 V=800.0 PL=0
MOVL C00910 V=800.0 PL=0
MOVL C00911 V=800.0 PL=0
MOVL C00912 V=800.0 PL=0
MOVL C00913 V=800.0 PL=0
MOVL C00914 V=800.0 PL=0
MOVL C00915 V=800.0 PL=0
MOVL C00916 V=800.0 PL=0
MOVL C00917 V=800.0 PL=0
MOVL C00918 V=800.0 PL=0
MOVL C00919 V=800.0 PL=0
MOVL C00920 V=800.0 PL=0
MOVL C00921 V=800.0 PL=0
MOVL C00922 V=800.0 PL=0
MOVL C00923 V=800.0 PL=0
MOVL C00924 V=800.0 PL=0
MOVL C00925 V=800.0 PL=0
MOVL C00926 V=800.0 PL=0
MOVL C00927 V=800.0 PL=0
MOVL C00928 V=800.0 PL=0
MOVL C00929 V=800.0 PL=0
MOVL C00930 V=800.0 PL=0
MOVL C00931 V=800.0 PL=0
MOVL C00932 V=800.0 PL=0
MOVL C00933 V=800.0 PL=0
MOVL C00934 V=800.0 PL=0
MOVL C00935 V=800.0 PL=0
MOVL C00936 V=800.0 PL=0
MOVL C00937 V=800.0 PL=0
MOVL C00938 V=800.0 PL=0
MOVL C00939 V=800.0 PL=0
MOVL C00940 V=800.0 PL=0
MOVL C00941 V=800.0 PL=0
MOVL C00942 V=800.0 PL=0
MOVL C00943 V=800.0 PL=0
MOVL C00944 V=800.0 PL=0
MOVL C00945 V=800.0 PL=0
MOVL C00946 V=800.0 PL=0
MOVL C00947 V=800.0 PL=0
MOVL C00948 V=800.0 PL=0
MOVL C00949 V=800.0 PL=0
MOVL C00950 V=800.0 PL=0
MOVL C00951 V=800.0 PL=0
MOVL C00952 V=800.0 PL=0
MOVL C00953 V=800.0 PL=0
MOVL C00954 V=800.0 PL=0
MOVL C00955 V=800.0 PL=0
MOVL C00956 V=800.0 PL=0
MOVL C00957 V=800.0 PL=0
MOVL C00958 V=800.0 PL=0
MOVL C00959 V=800.0 PL=0
MOVL C00960 V=800.0 PL=0
MOVL C00961 V=800.0 PL=0
MOVL C00962 V=800.0 PL=0
MOVL C00963 V=800.0 PL=0
MOVL C00964 V=800.0 PL=0
MOVL C00965 V=800.0 PL=0
MOVL C00966 V=800.0 PL=0
MOVL C00967 V=800.0 PL=0
MOVL C00968 V=800.0 PL=0
MOVL C00969 V=800.0 PL=0
MOVL C00970 V=800.0 PL=0
MOVL C00971 V=800.0 PL=0
MOVL C00972 V=800.0 PL=0
MOVL C00973 V=800.0 PL=0
MOVL C00974 V=800.0 PL=0
MOVL C00975 V=800.0 PL=0
MOVL C00976 V=800.0 PL=0
MOVL C00977 V=800.0 PL=0
MOVL C00978 V=800.0 PL=0
MOVL C00979 V=800.0 PL=0
MOVL C00980 V=800.0 PL=0
MOVL C00981 V=800.0 PL=0
MOVL C00982 V=800.0 PL=0
MOVL C00983 V=800.0 PL=0
MOVL C00984 V=800.0 PL=0
MOVL C00985 V=800.0 PL=0
MOVL C00986 V=800.0 PL=0
MOVL C00987 V=800.0 PL=0
MOVL C00988 V=800.0 PL=0
MOVL C00989 V=800.0 PL=0
MOVL C00990 V=800.0 PL=0
MOVL C00991 V=800.0 PL=0
MOVL C00992 V=800.0 PL=0
MOVL C00993 V=800.0 PL=0
MOVL C00994 V=800.0 PL=0
MOVL C00995 V=800.0 PL=0
MOVL C00996 V=800.0 PL=0
MOVL C00997 V=800.0 PL=0
MOVL C00998 V=800.0 PL=0
MOVL C00999 V=800.0 PL=0
MOVL C01000 V=800.0 PL=0
MOVL C01001 V=800.0 PL=0
MOVL C01002 V=800.0 PL=0
MOVL C01003 V=800.0 PL=0
MOVL C01004 V=800.0 PL=0
MOVL C01005 V=800.0 PL=0
MOVL C01006 V=800.0 PL=0
MOVL C01007 V=800.0 PL=0
MOVL C01008 V=800.0 PL=0
MOVL C01009 V=800.0 PL=0
MOVL C01010 V=800.0 PL=0
MOVL C01011 V=800.0 PL=0
MOVL C01012 V=800.0 PL=0
MOVL C01013 V=800.0 PL=0
MOVL C01014 V=800.0 PL=0
MOVL C01015 V=800.0 PL=0
MOVL C01016 V=800.0 PL=0
MOVL C01017 V=800.0 PL=0
MOVL C01018 V=800.0 PL=0
MOVL C01019 V=800.0 PL=0
MOVL C01020 V=800.0 PL=0
MOVL C01021 V=800.0 PL=0
MOVL C01022 V=800.0 PL=0
MOVL C01023 V=800.0 PL=0
MOVL C01024 V=800.0 PL=0
MOVL C01025 V=800.0 PL=0
MOVL C01026 V=800.0 PL=0
MOVL C01027 V=800.0 PL=0
MOVL C01028 V=800.0 PL=0
MOVL C01029 V=800.0 PL=0
MOVL C01030 V=800.0 PL=0
MOVL C01031 V=800.0 PL=0
MOVL C01032 V=800.0 PL=0
MOVL C01033 V=800.0 PL=0
MOVL C01034 V=800.0 PL=0
MOVL C01035 V=800.0 PL=0
MOVL C01036 V=800.0 PL=0
MOVL C01037 V=800.0 PL=0
MOVL C01038 V=800.0 PL=0
MOVL C01039 V=800.0 PL=0
MOVL C01040 V=800.0 PL=0
MOVL C01041 V=800.0 PL=0
MOVL C01042 V=800.0 PL=0
MOVL C01043 V=800.0 PL=0
MOVL C01044 V=800.0 PL=0
MOVL C01045 V=800.0 PL=0
MOVL C01046 V=800.0 PL=0
MOVL C01047 V=800.0 PL=0
MOVL C01048 V=800.0 PL=0
MOVL C01049 V=800.0 PL=0
MOVL C01050 V=800.0 PL=0
MOVL C01051 V=800.0 PL=0
MOVL C01052 V=800.0 PL=0
MOVL C01053 V=800.0 PL=0
MOVL C01054 V=800.0 PL=0
MOVL C01055 V=800.0 PL=0
MOVL C01056 V=800.0 PL=0
MOVL C01057 V=800.0 PL=0
MOVL C01058 V=800.0 PL=0
MOVL C01059 V=800.0 PL=0
MOVL C01060 V=800.0 PL=0
MOVL C01061 V=800.0 PL=0
MOVL C01062 V=800.0 PL=0
MOVL C01063 V=800.0 PL=0
MOVL C01064 V=800.0 PL=0
MOVL C01065 V=800.0 PL=0
MOVL C01066 V=800.0 PL=0
MOVL C01067 V=800.0 PL=0
MOVL C01068 V=800.0 PL=0
MOVL C01069 V=800.0 PL=0
MOVL C01070 V=800.0 PL=0
MOVL C01071 V=800.0 PL=0
MOVL C01072 V=800.0 PL=0
MOVL C01073 V=800.0 PL=0
MOVL C01074 V=800.0 PL=0
MOVL C01075 V=800.0 PL=0
MOVL C01076 V=800.0 PL=0
MOVL C01077 V=800.0 PL=0
MOVL C01078 V=800.0 PL=0
MOVL C01079 V=800.0 PL=0
MOVL C01080 V=800.0 PL=0
MOVL C01081 V=800.0 PL=0
MOVL C01082 V=800.0 PL=0
MOVL C01083 V=800.0 PL=0
MOVL C01084 V=800.0 PL=0
MOVL C01085 V=800.0 PL=0
MOVL C01086 V=800.0 PL=0
MOVL C01087 V=800.0 PL=0
MOVL C01088 V=800.0 PL=0
MOVL C01089 V=800.0 PL=0
MOVL C01090 V=800.0 PL=0
MOVL C01091 V=800.0 PL=0
MOVL C01092 V=800.0 PL=0
MOVL C01093 V=800.0 PL=0
MOVL C01094 V=800.0 PL=0
MOVL C01095 V=800.0 PL=0
MOVL C01096 V=800.0 PL=0
MOVL C01097 V=800.0 PL=0
MOVL C01098 V=800.0 PL=0
MOVL C01099 V=800.0 PL=0
MOVL C01100 V=800.0 PL=0
MOVL C01101 V=800.0 PL=0
MOVL C01102 V=800.0 PL=0
MOVL C01103 V=800.0 PL=0
MOVL C01104 V=800.0 PL=0
MOVL C01105 V=800.0 PL=0
MOVL C01106 V=800.0 PL=0
MOVL C01107 V=800.0 PL=0
MOVL C01108 V=800.0 PL=0
MOVL C01109 V=800.0 PL=0
MOVL C01110 V=800.0 PL=0
MOVL C01111 V=800.0 PL=0
MOVL C01112 V=800.0 PL=0
MOVL C01113 V=800.0 PL=0
MOVL C01114 V=800.0 PL=0
MOVL C01115 V=800.0 PL=0
MOVL C01116 V=800.0 PL=0
MOVL C01117 V=800.0 PL=0
MOVL C01118 V=800.0 PL=0
MOVL C01119 V=800.0 PL=0
MOVL C01120 V=800.0 PL=0
MOVL C01121 V=800.0 PL=0
MOVL C01122 V=800.0 PL=0
MOVL C01123 V=800.0 PL=0
MOVL C01124 V=800.0 PL=0
MOVL C01125 V=800.0 PL=0
MOVL C01126 V=800.0 PL=0
MOVL C01127 V=800.0 PL=0
MOVL C01128 V=800.0 PL=0
MOVL C01129 V=800.0 PL=0
MOVL C01130 V=800.0 PL=0
MOVL C01131 V=800.0 PL=0
MOVL C01132 V=800.0 PL=0
MOVL C01133 V=800.0 PL=0
MOVL C01134 V=800.0 PL=0
MOVL C01135 V=800.0 PL=0
MOVL C01136 V=800.0 PL=0
MOVL C01137 V=800.0 PL=0
MOVL C01138 V=800.0 PL=0
MOVL C01139 V=800.0 PL=0
MOVL C01140 V=800.0 PL=0
MOVL C01141 V=800.0 PL=0
MOVL C01142 V=800.0 PL=0
MOVL C01143 V=800.0 PL=0
MOVL C01144 V=800.0 PL=0
MOVL C01145 V=800.0 PL=0
MOVL C01146 V=800.0 PL=0
MOVL C01147 V=800.0 PL=0
MOVL C01148 V=800.0 PL=0
MOVL C01149 V=800.0 PL=0
MOVL C01150 V=800.0 PL=0
MOVL C01151 V=800.0 PL=0
MOVL C01152 V=800.0 PL=0
MOVL C01153 V=800.0 PL=0
MOVL C01154 V=800.0 PL=0
MOVL C01155 V=800.0 PL=0
MOVL C01156 V=800.0 PL=0
MOVL C01157 V=800.0 PL=0
MOVL C01158 V=800.0 PL=0
MOVL C01159 V=800.0 PL=0
MOVL C01160 V=800.0 PL=0
MOVL C01161 V=800.0 PL=0
MOVL C01162 V=800.0 PL=0
MOVL C01163 V=800.0 PL=0
MOVL C01164 V=800.0 PL=0
MOVL C01165 V=800.0 PL=0
MOVL C01166 V=800.0 PL=0
MOVL C01167 V=800.0 PL=0
MOVL C01168 V=800.0 PL=0
MOVL C01169 V=800.0 PL=0
MOVL C01170 V=800.0 PL=0
MOVL C01171 V=800.0 PL=0
MOVL C01172 V=800.0 PL=0
MOVL C01173 V=800.0 PL=0
MOVL C01174 V=800.0 PL=0
MOVL C01175 V=800.0 PL=0
MOVL C01176 V=800.0 PL=0
MOVL C01177 V=800.0 PL=0
MOVL C01178 V=800.0 PL=0
MOVL C01179 V=800.0 PL=0
MOVL C01180 V=800.0 PL=0
MOVL C01181 V=800.0 PL=0
MOVL C01182 V=800.0 PL=0
MOVL C01183 V=800.0 PL=0
MOVL C01184 V=800.0 PL=0
MOVL C01185 V=800.0 PL=0
MOVL C01186 V=800.0 PL=0
MOVL C01187 V=800.0 PL=0
MOVL C01188 V=800.0 PL=0
MOVL C01189 V=800.0 PL=0
MOVL C01190 V=800.0 PL=0
MOVL C01191 V=800.0 PL=0
MOVL C01192 V=800.0 PL=0
MOVL C01193 V=800.0 PL=0
MOVL C01194 V=800.0 PL=0
MOVL C01195 V=800.0 PL=0
MOVL C01196 V=800.0 PL=0
MOVL C01197 V=800.0 PL=0
MOVL C01198 V=800.0 PL=0
MOVL C01199 V=800.0 PL=0
MOVL C01200 V=800.0 PL=0
MOVL C01201 V=800.0 PL=0
MOVL C01202 V=800.0 PL=0
MOVL C01203 V=800.0 PL=0
MOVL C01204 V=800.0 PL=0
MOVL C01205 V=800.0 PL=0
MOVL C01206 V=800.0 PL=0
MOVL C01207 V=800.0 PL=0
MOVL C01208 V=800.0 PL=0
MOVL C01209 V=800.0 PL=0
MOVL C01210 V=800.0 PL=0
MOVL C01211 V=800.0 PL=0
MOVL C01212 V=800.0 PL=0
MOVL C01213 V=800.0 PL=0
MOVL C01214 V=800.0 PL=0
MOVL C01215 V=800.0 PL=0
MOVL C01216 V=800.0 PL=0
MOVL C01217 V=800.0 PL=0
MOVL C01218 V=800.0 PL=0
MOVL C01219 V=800.0 PL=0
MOVL C01220 V=800.0 PL=0
MOVL C01221 V=800.0 PL=0
MOVL C01222 V=800.0 PL=0
MOVL C01223 V=800.0 PL=0
MOVL C01224 V=800.0 PL=0
MOVL C01225 V=800.0 PL=0
MOVL C01226 V=800.0 PL=0
MOVL C01227 V=800.0 PL=0
MOVL C01228 V=800.0 PL=0
MOVL C01229 V=800.0 PL=0
MOVL C01230 V=800.0 PL=0
MOVL C01231 V=800.0 PL=0
MOVL C01232 V=800.0 PL=0
MOVL C01233 V=800.0 PL=0
MOVL C01234 V=800.0 PL=0
MOVL C01235 V=800.0 PL=0
MOVL C01236 V=800.0 PL=0
MOVL C01237 V=800.0 PL=0
MOVL C01238 V=800.0 PL=0
MOVL C01239 V=800.0 PL=0
MOVL C01240 V=800.0 PL=0
MOVL C01241 V=800.0 PL=0
MOVL C01242 V=800.0 PL=0
MOVL C01243 V=800.0 PL=0
MOVL C01244 V=800.0 PL=0
MOVL C01245 V=800.0 PL=0
MOVL C01246 V=800.0 PL=0
MOVL C01247 V=800.0 PL=0
MOVL C01248 V=800.0 PL=0
MOVL C01249 V=800.0 PL=0
MOVL C01250 V=800.0 PL=0
MOVL C01251 V=800.0 PL=0
MOVL C01252 V=800.0 PL=0
MOVL C01253 V=800.0 PL=0
MOVL C01254 V=800.0 PL=0
MOVL C01255 V=800.0 PL=0
MOVL C01256 V=800.0 PL=0
MOVL C01257 V=800.0 PL=0
MOVL C01258 V=800.0 PL=0
MOVL C01259 V=800.0 PL=0
MOVL C01260 V=800.0 PL=0
MOVL C01261 V=800.0 PL=0
MOVL C01262 V=800.0 PL=0
MOVL C01263 V=800.0 PL=0
MOVL C01264 V=800.0 PL=0
MOVL C01265 V=800.0 PL=0
MOVL C01266 V=800.0 PL=0
MOVL C01267 V=800.0 PL=0
MOVL C01268 V=800.0 PL=0
MOVL C01269 V=800.0 PL=0
MOVL C01270 V=800.0 PL=0
MOVL C01271 V=800.0 PL=0
MOVL C01272 V=800.0 PL=0
MOVL C01273 V=800.0 PL=0
MOVL C01274 V=800.0 PL=0
MOVL C01275 V=800.0 PL=0
MOVL C01276 V=800.0 PL=0
MOVL C01277 V=800.0 PL=0
MOVL C01278 V=800.0 PL=0
MOVL C01279 V=800.0 PL=0
MOVL C01280 V=800.0 PL=0
MOVL C01281 V=800.0 PL=0
MOVL C01282 V=800.0 PL=0
MOVL C01283 V=800.0 PL=0
MOVL C01284 V=800.0 PL=0
MOVL C01285 V=800.0 PL=0
MOVL C01286 V=800.0 PL=0
MOVL C01287 V=800.0 PL=0
MOVL C01288 V=800.0 PL=0
MOVL C01289 V=800.0 PL=0
MOVL C01290 V=800.0 PL=0
MOVL C01291 V=800.0 PL=0
MOVL C01292 V=800.0 PL=0
MOVL C01293 V=800.0 PL=0
MOVL C01294 V=800.0 PL=0
MOVL C01295 V=800.0 PL=0
MOVL C01296 V=800.0 PL=0
MOVL C01297 V=800.0 PL=0
MOVL C01298 V=800.0 PL=0
MOVL C01299 V=800.0 PL=0
MOVL C01300 V=800.0 PL=0
MOVL C01301 V=800.0 PL=0
MOVL C01302 V=800.0 PL=0
MOVL C01303 V=800.0 PL=0
MOVL C01304 V=800.0 PL=0
MOVL C01305 V=800.0 PL=0
MOVL C01306 V=800.0 PL=0
MOVL C01307 V=800.0 PL=0
MOVL C01308 V=800.0 PL=0
MOVL C01309 V=800.0 PL=0
MOVL C01310 V=800.0 PL=0
MOVL C01311 V=800.0 PL=0
MOVL C01312 V=800.0 PL=0
MOVL C01313 V=800.0 PL=0
MOVL C01314 V=800.0 PL=0
MOVL C01315 V=800.0 PL=0
MOVL C01316 V=800.0 PL=0
MOVL C01317 V=800.0 PL=0
MOVL C01318 V=800.0 PL=0
MOVL C01319 V=800.0 PL=0
MOVL C01320 V=800.0 PL=0
MOVL C01321 V=800.0 PL=0
MOVL C01322 V=800.0 PL=0
MOVL C01323 V=800.0 PL=0
MOVL C01324 V=800.0 PL=0
MOVL C01325 V=800.0 PL=0
MOVL C01326 V=800.0 PL=0
MOVL C01327 V=800.0 PL=0
MOVL C01328 V=800.0 PL=0
MOVL C01329 V=800.0 PL=0
MOVL C01330 V=800.0 PL=0
MOVL C01331 V=800.0 PL=0
MOVL C01332 V=800.0 PL=0
MOVL C01333 V=800.0 PL=0
MOVL C01334 V=800.0 PL=0
MOVL C01335 V=800.0 PL=0
MOVL C01336 V=800.0 PL=0
MOVL C01337 V=800.0 PL=0
MOVL C01338 V=800.0 PL=0
MOVL C01339 V=800.0 PL=0
MOVL C01340 V=800.0 PL=0
MOVL C01341 V=800.0 PL=0
MOVL C01342 V=800.0 PL=0
MOVL C01343 V=800.0 PL=0
MOVL C01344 V=800.0 PL=0
MOVL C01345 V=800.0 PL=0
MOVL C01346 V=800.0 PL=0
MOVL C01347 V=800.0 PL=0
MOVL C01348 V=800.0 PL=0
MOVL C01349 V=800.0 PL=0
MOVL C01350 V=800.0 PL=0
MOVL C01351 V=800.0 PL=0
MOVL C01352 V=800.0 PL=0
MOVL C01353 V=800.0 PL=0
MOVL C01354 V=800.0 PL=0
MOVL C01355 V=800.0 PL=0
MOVL C01356 V=800.0 PL=0
MOVL C01357 V=800.0 PL=0
MOVL C01358 V=800.0 PL=0
MOVL C01359 V=800.0 PL=0
MOVL C01360 V=800.0 PL=0
MOVL C01361 V=800.0 PL=0
MOVL C01362 V=800.0 PL=0
MOVL C01363 V=800.0 PL=0
MOVL C01364 V=800.0 PL=0
MOVL C01365 V=800.0 PL=0
MOVL C01366 V=800.0 PL=0
MOVL C01367 V=800.0 PL=0
MOVL C01368 V=800.0 PL=0
MOVL C01369 V=800.0 PL=0
MOVL C01370 V=800.0 PL=0
MOVL C01371 V=800.0 PL=0
MOVL C01372 V=800.0 PL=0
MOVL C01373 V=800.0 PL=0
MOVL C01374 V=800.0 PL=0
MOVL C01375 V=800.0 PL=0
MOVL C01376 V=800.0 PL=0
MOVL C01377 V=800.0 PL=0
MOVL C01378 V=800.0 PL=0
MOVL C01379 V=800.0 PL=0
MOVL C01380 V=800.0 PL=0
MOVL C01381 V=800.0 PL=0
MOVL C01382 V=800.0 PL=0
MOVL C01383 V=800.0 PL=0
MOVL C01384 V=800.0 PL=0
MOVL C01385 V=800.0 PL=0
MOVL C01386 V=800.0 PL=0
MOVL C01387 V=800.0 PL=0
MOVL C01388 V=800.0 PL=0
MOVL C01389 V=800.0 PL=0
MOVL C01390 V=800.0 PL=0
MOVL C01391 V=800.0 PL=0
MOVL C01392 V=800.0 PL=0
MOVL C01393 V=800.0 PL=0
MOVL C01394 V=800.0 PL=0
MOVL C01395 V=800.0 PL=0
MOVL C01396 V=800.0 PL=0
MOVL C01397 V=800.0 PL=0
MOVL C01398 V=800.0 PL=0
MOVL C01399 V=800.0 PL=0
MOVL C01400 V=800.0 PL=0
MOVL C01401 V=800.0 PL=0
MOVL C01402 V=800.0 PL=0
MOVL C01403 V=800.0 PL=0
MOVL C01404 V=800.0 PL=0
MOVL C01405 V=800.0 PL=0
MOVL C01406 V=800.0 PL=0
MOVL C01407 V=800.0 PL=0
MOVL C01408 V=800.0 PL=0
MOVL C01409 V=800.0 PL=0
MOVL C01410 V=800.0 PL=0
MOVL C01411 V=800.0 PL=0
MOVL C01412 V=800.0 PL=0
MOVL C01413 V=800.0 PL=0
MOVL C01414 V=800.0 PL=0
MOVL C01415 V=800.0 PL=0
MOVL C01416 V=800.0 PL=0
MOVL C01417 V=800.0 PL=0
MOVL C01418 V=800.0 PL=0
MOVL C01419 V=800.0 PL=0
MOVL C01420 V=800.0 PL=0
MOVL C01421 V=800.0 PL=0
MOVL C01422 V=800.0 PL=0
MOVL C01423 V=800.0 PL=0
MOVL C01424 V=800.0 PL=0
MOVL C01425 V=800.0 PL=0
MOVL C01426 V=800.0 PL=0
MOVL C01427 V=800.0 PL=0
MOVL C01428 V=800.0 PL=0
MOVL C01429 V=800.0 PL=0
MOVL C01430 V=800.0 PL=0
MOVL C01431 V=800.0 PL=0
MOVL C01432 V=800.0 PL=0
MOVL C01433 V=800.0 PL=0
MOVL C01434 V=800.0 PL=0
MOVL C01435 V=800.0 PL=0
MOVL C01436 V=800.0 PL=0
MOVL C01437 V=800.0 PL=0
MOVL C01438 V=800.0 PL=0
MOVL C01439 V=800.0 PL=0
MOVL C01440 V=800.0 PL=0
MOVL C01441 V=800.0 PL=0
MOVL C01442 V=800.0 PL=0
MOVL C01443 V=800.0 PL=0
MOVL C01444 V=800.0 PL=0
MOVL C01445 V=800.0 PL=0
MOVL C01446 V=800.0 PL=0
MOVL C01447 V=800.0 PL=0
MOVL C01448 V=800.0 PL=0
MOVL C01449 V=800.0 PL=0
MOVL C01450 V=800.0 PL=0
MOVL C01451 V=800.0 PL=0
MOVL C01452 V=800.0 PL=0
MOVL C01453 V=800.0 PL=0
MOVL C01454 V=800.0 PL=0
MOVL C01455 V=800.0 PL=0
MOVL C01456 V=800.0 PL=0
MOVL C01457 V=800.0 PL=0
MOVL C01458 V=800.0 PL=0
MOVL C01459 V=800.0 PL=0
MOVL C01460 V=800.0 PL=0
MOVL C01461 V=800.0 PL=0
MOVL C01462 V=800.0 PL=0
MOVL C01463 V=800.0 PL=0
MOVL C01464 V=800.0 PL=0
MOVL C01465 V=800.0 PL=0
MOVL C01466 V=800.0 PL=0
MOVL C01467 V=800.0 PL=0
MOVL C01468 V=800.0 PL=0
MOVL C01469 V=800.0 PL=0
MOVL C01470 V=800.0 PL=0
MOVL C01471 V=800.0 PL=0
MOVL C01472 V=800.0 PL=0
MOVL C01473 V=800.0 PL=0
MOVL C01474 V=800.0 PL=0
MOVL C01475 V=800.0 PL=0
MOVL C01476 V=800.0 PL=0
MOVL C01477 V=800.0 PL=0
MOVL C01478 V=800.0 PL=0
MOVL C01479 V=800.0 PL=0
MOVL C01480 V=800.0 PL=0
MOVL C01481 V=800.0 PL=0
MOVL C01482 V=800.0 PL=0
MOVL C01483 V=800.0 PL=0
MOVL C01484 V=800.0 PL=0
MOVL C01485 V=800.0 PL=0
MOVL C01486 V=800.0 PL=0
MOVL C01487 V=800.0 PL=0
MOVL C01488 V=800.0 PL=0
MOVL C01489 V=800.0 PL=0
MOVL C01490 V=800.0 PL=0
MOVL C01491 V=800.0 PL=0
MOVL C01492 V=800.0 PL=0
MOVL C01493 V=800.0 PL=0
MOVL C01494 V=800.0 PL=0
MOVL C01495 V=800.0 PL=0
MOVL C01496 V=800.0 PL=0
MOVL C01497 V=800.0 PL=0
MOVL C01498 V=800.0 PL=0
MOVL C01499 V=800.0 PL=0
MOVL C01500 V=800.0 PL=0
MOVL C01501 V=800.0 PL=0
MOVL C01502 V=800.0 PL=0
MOVL C01503 V=800.0 PL=0
MOVL C01504 V=800.0 PL=0
MOVL C01505 V=800.0 PL=0
MOVL C01506 V=800.0 PL=0
MOVL C01507 V=800.0 PL=0
MOVL C01508 V=800.0 PL=0
MOVL C01509 V=800.0 PL=0
MOVL C01510 V=800.0 PL=0
MOVL C01511 V=800.0 PL=0
MOVL C01512 V=800.0 PL=0
MOVL C01513 V=800.0 PL=0
MOVL C01514 V=800.0 PL=0
MOVL C01515 V=800.0 PL=0
MOVL C01516 V=800.0 PL=0
MOVL C01517 V=800.0 PL=0
MOVL C01518 V=800.0 PL=0
MOVL C01519 V=800.0 PL=0
MOVL C01520 V=800.0 PL=0
MOVL C01521 V=800.0 PL=0
MOVL C01522 V=800.0 PL=0
MOVL C01523 V=800.0 PL=0
MOVL C01524 V=800.0 PL=0
MOVL C01525 V=800.0 PL=0
MOVL C01526 V=800.0 PL=0
MOVL C01527 V=800.0 PL=0
MOVL C01528 V=800.0 PL=0
MOVL C01529 V=800.0 PL=0
MOVL C01530 V=800.0 PL=0
MOVL C01531 V=800.0 PL=0
MOVL C01532 V=800.0 PL=0
MOVL C01533 V=800.0 PL=0
MOVL C01534 V=800.0 PL=0
MOVL C01535 V=800.0 PL=0
MOVL C01536 V=800.0 PL=0
MOVL C01537 V=800.0 PL=0
MOVL C01538 V=800.0 PL=0
MOVL C01539 V=800.0 PL=0
MOVL C01540 V=800.0 PL=0
MOVL C01541 V=800.0 PL=0
MOVL C01542 V=800.0 PL=0
MOVL C01543 V=800.0 PL=0
MOVL C01544 V=800.0 PL=0
MOVL C01545 V=800.0 PL=0
MOVL C01546 V=800.0 PL=0
MOVL C01547 V=800.0 PL=0
MOVL C01548 V=800.0 PL=0
MOVL C01549 V=800.0 PL=0
MOVL C01550 V=800.0 PL=0
MOVL C01551 V=800.0 PL=0
MOVL C01552 V=800.0 PL=0
MOVL C01553 V=800.0 PL=0
MOVL C01554 V=800.0 PL=0
MOVL C01555 V=800.0 PL=0
MOVL C01556 V=800.0 PL=0
MOVL C01557 V=800.0 PL=0
MOVL C01558 V=800.0 PL=0
MOVL C01559 V=800.0 PL=0
MOVL C01560 V=800.0 PL=0
MOVL C01561 V=800.0 PL=0
MOVL C01562 V=800.0 PL=0
MOVL C01563 V=800.0 PL=0
MOVL C01564 V=800.0 PL=0
MOVL C01565 V=800.0 PL=0
MOVL C01566 V=800.0 PL=0
MOVL C01567 V=800.0 PL=0
MOVL C01568 V=800.0 PL=0
MOVL C01569 V=800.0 PL=0
MOVL C01570 V=800.0 PL=0
MOVL C01571 V=800.0 PL=0
MOVL C01572 V=800.0 PL=0
MOVL C01573 V=800.0 PL=0
MOVL C01574 V=800.0 PL=0
MOVL C01575 V=800.0 PL=0
MOVL C01576 V=800.0 PL=0
MOVL C01577 V=800.0 PL=0
MOVL C01578 V=800.0 PL=0
MOVL C01579 V=800.0 PL=0
MOVL C01580 V=800.0 PL=0
MOVL C01581 V=800.0 PL=0
MOVL C01582 V=800.0 PL=0
MOVL C01583 V=800.0 PL=0
MOVL C01584 V=800.0 PL=0
MOVL C01585 V=800.0 PL=0
MOVL C01586 V=800.0 PL=0
MOVL C01587 V=800.0 PL=0
MOVL C01588 V=800.0 PL=0
MOVL C01589 V=800.0 PL=0
MOVL C01590 V=800.0 PL=0
MOVL C01591 V=800.0 PL=0
MOVL C01592 V=800.0 PL=0
MOVL C01593 V=800.0 PL=0
MOVL C01594 V=800.0 PL=0
MOVL C01595 V=800.0 PL=0
MOVL C01596 V=800.0 PL=0
MOVL C01597 V=800.0 PL=0
MOVL C01598 V=800.0 PL=0
MOVL C01599 V=800.0 PL=0
MOVL C01600 V=800.0 PL=0
MOVL C01601 V=800.0 PL=0
MOVL C01602 V=800.0 PL=0
MOVL C01603 V=800.0 PL=0
MOVL C01604 V=800.0 PL=0
MOVL C01605 V=800.0 PL=0
MOVL C01606 V=800.0 PL=0
MOVL C01607 V=800.0 PL=0
MOVL C01608 V=800.0 PL=0
MOVL C01609 V=800.0 PL=0
MOVL C01610 V=800.0 PL=0
MOVL C01611 V=800.0 PL=0
MOVL C01612 V=800.0 PL=0
MOVL C01613 V=800.0 PL=0
MOVL C01614 V=800.0 PL=0
MOVL C01615 V=800.0 PL=0
MOVL C01616 V=800.0 PL=0
MOVL C01617 V=800.0 PL=0
MOVL C01618 V=800.0 PL=0
MOVL C01619 V=800.0 PL=0
MOVL C01620 V=800.0 PL=0
MOVL C01621 V=800.0 PL=0
MOVL C01622 V=800.0 PL=0
MOVL C01623 V=800.0 PL=0
MOVL C01624 V=800.0 PL=0
MOVL C01625 V=800.0 PL=0
MOVL C01626 V=800.0 PL=0
MOVL C01627 V=800.0 PL=0
MOVL C01628 V=800.0 PL=0
MOVL C01629 V=800.0 PL=0
MOVL C01630 V=800.0 PL=0
MOVL C01631 V=800.0 PL=0
MOVL C01632 V=800.0 PL=0
MOVL C01633 V=800.0 PL=0
MOVL C01634 V=800.0 PL=0
MOVL C01635 V=800.0 PL=0
MOVL C01636 V=800.0 PL=0
MOVL C01637 V=800.0 PL=0
MOVL C01638 V=800.0 PL=0
MOVL C01639 V=800.0 PL=0
MOVL C01640 V=800.0 PL=0
MOVL C01641 V=800.0 PL=0
MOVL C01642 V=800.0 PL=0
MOVL C01643 V=800.0 PL=0
MOVL C01644 V=800.0 PL=0
MOVL C01645 V=800.0 PL=0
MOVL C01646 V=800.0 PL=0
MOVL C01647 V=800.0 PL=0
MOVL C01648 V=800.0 PL=0
MOVL C01649 V=800.0 PL=0
MOVL C01650 V=800.0 PL=0
MOVL C01651 V=800.0 PL=0
MOVL C01652 V=800.0 PL=0
MOVL C01653 V=800.0 PL=0
MOVL C01654 V=800.0 PL=0
MOVL C01655 V=800.0 PL=0
MOVL C01656 V=800.0 PL=0
MOVL C01657 V=800.0 PL=0
MOVL C01658 V=800.0 PL=0
MOVL C01659 V=800.0 PL=0
MOVL C01660 V=800.0 PL=0
MOVL C01661 V=800.0 PL=0
MOVL C01662 V=800.0 PL=0
MOVL C01663 V=800.0 PL=0
MOVL C01664 V=800.0 PL=0
MOVL C01665 V=800.0 PL=0
MOVL C01666 V=800.0 PL=0
MOVL C01667 V=800.0 PL=0
MOVL C01668 V=800.0 PL=0
MOVL C01669 V=800.0 PL=0
MOVL C01670 V=800.0 PL=0
MOVL C01671 V=800.0 PL=0
MOVL C01672 V=800.0 PL=0
MOVL C01673 V=800.0 PL=0
MOVL C01674 V=800.0 PL=0
MOVL C01675 V=800.0 PL=0
MOVL C01676 V=800.0 PL=0
MOVL C01677 V=800.0 PL=0
MOVL C01678 V=800.0 PL=0
MOVL C01679 V=800.0 PL=0
MOVL C01680 V=800.0 PL=0
MOVL C01681 V=800.0 PL=0
MOVL C01682 V=800.0 PL=0
MOVL C01683 V=800.0 PL=0
MOVL C01684 V=800.0 PL=0
MOVL C01685 V=800.0 PL=0
MOVL C01686 V=800.0 PL=0
MOVL C01687 V=800.0 PL=0
MOVL C01688 V=800.0 PL=0
MOVL C01689 V=800.0 PL=0
MOVL C01690 V=800.0 PL=0
MOVL C01691 V=800.0 PL=0
MOVL C01692 V=800.0 PL=0
MOVL C01693 V=800.0 PL=0
MOVL C01694 V=800.0 PL=0
MOVL C01695 V=800.0 PL=0
MOVL C01696 V=800.0 PL=0
MOVL C01697 V=800.0 PL=0
MOVL C01698 V=800.0 PL=0
MOVL C01699 V=800.0 PL=0
MOVL C01700 V=800.0 PL=0
MOVL C01701 V=800.0 PL=0
MOVL C01702 V=800.0 PL=0
MOVL C01703 V=800.0 PL=0
MOVL C01704 V=800.0 PL=0
MOVL C01705 V=800.0 PL=0
MOVL C01706 V=800.0 PL=0
MOVL C01707 V=800.0 PL=0
MOVL C01708 V=800.0 PL=0
MOVL C01709 V=800.0 PL=0
MOVL C01710 V=800.0 PL=0
MOVL C01711 V=800.0 PL=0
MOVL C01712 V=800.0 PL=0
MOVL C01713 V=800.0 PL=0
MOVL C01714 V=800.0 PL=0
MOVL C01715 V=800.0 PL=0
MOVL C01716 V=800.0 PL=0
MOVL C01717 V=800.0 PL=0
MOVL C01718 V=800.0 PL=0
MOVL C01719 V=800.0 PL=0
MOVL C01720 V=800.0 PL=0
MOVL C01721 V=800.0 PL=0
MOVL C01722 V=800.0 PL=0
MOVL C01723 V=800.0 PL=0
MOVL C01724 V=800.0 PL=0
MOVL C01725 V=800.0 PL=0
MOVL C01726 V=800.0 PL=0
MOVL C01727 V=800.0 PL=0
MOVL C01728 V=800.0 PL=0
MOVL C01729 V=800.0 PL=0
MOVL C01730 V=800.0 PL=0
MOVL C01731 V=800.0 PL=0
MOVL C01732 V=800.0 PL=0
MOVL C01733 V=800.0 PL=0
MOVL C01734 V=800.0 PL=0
MOVL C01735 V=800.0 PL=0
MOVL C01736 V=800.0 PL=0
MOVL C01737 V=800.0 PL=0
MOVL C01738 V=800.0 PL=0
MOVL C01739 V=800.0 PL=0
MOVL C01740 V=800.0 PL=0
MOVL C01741 V=800.0 PL=0
MOVL C01742 V=800.0 PL=0
MOVL C01743 V=800.0 PL=0
MOVL C01744 V=800.0 PL=0
MOVL C01745 V=800.0 PL=0
MOVL C01746 V=800.0 PL=0
MOVL C01747 V=800.0 PL=0
MOVL C01748 V=800.0 PL=0
MOVL C01749 V=800.0 PL=0
MOVL C01750 V=800.0 PL=0
MOVL C01751 V=800.0 PL=0
MOVL C01752 V=800.0 PL=0
MOVL C01753 V=800.0 PL=0
MOVL C01754 V=800.0 PL=0
MOVL C01755 V=800.0 PL=0
MOVL C01756 V=800.0 PL=0
MOVL C01757 V=800.0 PL=0
MOVL C01758 V=800.0 PL=0
MOVL C01759 V=800.0 PL=0
MOVL C01760 V=800.0 PL=0
MOVL C01761 V=800.0 PL=0
MOVL C01762 V=800.0 PL=0
MOVL C01763 V=800.0 PL=0
MOVL C01764 V=800.0 PL=0
MOVL C01765 V=800.0 PL=0
MOVL C01766 V=800.0 PL=0
MOVL C01767 V=800.0 PL=0
MOVL C01768 V=800.0 PL=0
MOVL C01769 V=800.0 PL=0
MOVL C01770 V=800.0 PL=0
MOVL C01771 V=800.0 PL=0
MOVL C01772 V=800.0 PL=0
MOVL C01773 V=800.0 PL=0
MOVL C01774 V=800.0 PL=0
MOVL C01775 V=800.0 PL=0
MOVL C01776 V=800.0 PL=0
MOVL C01777 V=800.0 PL=0
MOVL C01778 V=800.0 PL=0
MOVL C01779 V=800.0 PL=0
MOVL C01780 V=800.0 PL=0
MOVL C01781 V=800.0 PL=0
MOVL C01782 V=800.0 PL=0
MOVL C01783 V=800.0 PL=0
MOVL C01784 V=800.0 PL=0
MOVL C01785 V=800.0 PL=0
MOVL C01786 V=800.0 PL=0
MOVL C01787 V=800.0 PL=0
MOVL C01788 V=800.0 PL=0
MOVL C01789 V=800.0 PL=0
MOVL C01790 V=800.0 PL=0
MOVL C01791 V=800.0 PL=0
MOVL C01792 V=800.0 PL=0
MOVL C01793 V=800.0 PL=0
MOVL C01794 V=800.0 PL=0
MOVL C01795 V=800.0 PL=0
MOVL C01796 V=800.0 PL=0
MOVL C01797 V=800.0 PL=0
MOVL C01798 V=800.0 PL=0
MOVL C01799 V=800.0 PL=0
MOVL C01800 V=800.0 PL=0
MOVL C01801 V=800.0 PL=0
MOVL C01802 V=800.0 PL=0
MOVL C01803 V=800.0 PL=0
MOVL C01804 V=800.0 PL=0
MOVL C01805 V=800.0 PL=0
MOVL C01806 V=800.0 PL=0
MOVL C01807 V=800.0 PL=0
MOVL C01808 V=800.0 PL=0
MOVL C01809 V=800.0 PL=0
MOVL C01810 V=800.0 PL=0
MOVL C01811 V=800.0 PL=0
MOVL C01812 V=800.0 PL=0
MOVL C01813 V=800.0 PL=0
MOVL C01814 V=800.0 PL=0
MOVL C01815 V=800.0 PL=0
MOVL C01816 V=800.0 PL=0
MOVL C01817 V=800.0 PL=0
MOVL C01818 V=800.0 PL=0
MOVL C01819 V=800.0 PL=0
MOVL C01820 V=800.0 PL=0
MOVL C01821 V=800.0 PL=0
MOVL C01822 V=800.0 PL=0
MOVL C01823 V=800.0 PL=0
MOVL C01824 V=800.0 PL=0
MOVL C01825 V=800.0 PL=0
MOVL C01826 V=800.0 PL=0
MOVL C01827 V=800.0 PL=0
MOVL C01828 V=800.0 PL=0
MOVL C01829 V=800.0 PL=0
MOVL C01830 V=800.0 PL=0
MOVL C01831 V=800.0 PL=0
MOVL C01832 V=800.0 PL=0
MOVL C01833 V=800.0 PL=0
MOVL C01834 V=800.0 PL=0
MOVL C01835 V=800.0 PL=0
MOVL C01836 V=800.0 PL=0
MOVL C01837 V=800.0 PL=0
MOVL C01838 V=800.0 PL=0
MOVL C01839 V=800.0 PL=0
MOVL C01840 V=800.0 PL=0
MOVL C01841 V=800.0 PL=0
MOVL C01842 V=800.0 PL=0
MOVL C01843 V=800.0 PL=0
MOVL C01844 V=800.0 PL=0
MOVL C01845 V=800.0 PL=0
MOVL C01846 V=800.0 PL=0
MOVL C01847 V=800.0 PL=0
MOVL C01848 V=800.0 PL=0
MOVL C01849 V=800.0 PL=0
MOVL C01850 V=800.0 PL=0
MOVL C01851 V=800.0 PL=0
MOVL C01852 V=800.0 PL=0
MOVL C01853 V=800.0 PL=0
MOVL C01854 V=800.0 PL=0
MOVL C01855 V=800.0 PL=0
MOVL C01856 V=800.0 PL=0
MOVL C01857 V=800.0 PL=0
MOVL C01858 V=800.0 PL=0
MOVL C01859 V=800.0 PL=0
MOVL C01860 V=800.0 PL=0
MOVL C01861 V=800.0 PL=0
MOVL C01862 V=800.0 PL=0
MOVL C01863 V=800.0 PL=0
MOVL C01864 V=800.0 PL=0
MOVL C01865 V=800.0 PL=0
MOVL C01866 V=800.0 PL=0
MOVL C01867 V=800.0 PL=0
MOVL C01868 V=800.0 PL=0
MOVL C01869 V=800.0 PL=0
MOVL C01870 V=800.0 PL=0
MOVL C01871 V=800.0 PL=0
MOVL C01872 V=800.0 PL=0
MOVL C01873 V=800.0 PL=0
MOVL C01874 V=800.0 PL=0
MOVL C01875 V=800.0 PL=0
MOVL C01876 V=800.0 PL=0
MOVL C01877 V=800.0 PL=0
MOVL C01878 V=800.0 PL=0
MOVL C01879 V=800.0 PL=0
MOVL C01880 V=800.0 PL=0
MOVL C01881 V=800.0 PL=0
MOVL C01882 V=800.0 PL=0
MOVL C01883 V=800.0 PL=0
MOVL C01884 V=800.0 PL=0
MOVL C01885 V=800.0 PL=0
MOVL C01886 V=800.0 PL=0
MOVL C01887 V=800.0 PL=0
MOVL C01888 V=800.0 PL=0
MOVL C01889 V=800.0 PL=0
MOVL C01890 V=800.0 PL=0
MOVL C01891 V=800.0 PL=0
MOVL C01892 V=800.0 PL=0
MOVL C01893 V=800.0 PL=0
MOVL C01894 V=800.0 PL=0
MOVL C01895 V=800.0 PL=0
MOVL C01896 V=800.0 PL=0
MOVL C01897 V=800.0 PL=0
MOVL C01898 V=800.0 PL=0
MOVL C01899 V=800.0 PL=0
MOVL C01900 V=800.0 PL=0
MOVL C01901 V=800.0 PL=0
MOVL C01902 V=800.0 PL=0
MOVL C01903 V=800.0 PL=0
MOVL C01904 V=800.0 PL=0
MOVL C01905 V=800.0 PL=0
MOVL C01906 V=800.0 PL=0
MOVL C01907 V=800.0 PL=0
MOVL C01908 V=800.0 PL=0
MOVL C01909 V=800.0 PL=0
MOVL C01910 V=800.0 PL=0
MOVL C01911 V=800.0 PL=0
MOVL C01912 V=800.0 PL=0
MOVL C01913 V=800.0 PL=0
MOVL C01914 V=800.0 PL=0
MOVL C01915 V=800.0 PL=0
MOVL C01916 V=800.0 PL=0
MOVL C01917 V=800.0 PL=0
MOVL C01918 V=800.0 PL=0
MOVL C01919 V=800.0 PL=0
MOVL C01920 V=800.0 PL=0
MOVL C01921 V=800.0 PL=0
MOVL C01922 V=800.0 PL=0
MOVL C01923 V=800.0 PL=0
MOVL C01924 V=800.0 PL=0
MOVL C01925 V=800.0 PL=0
MOVL C01926 V=800.0 PL=0
MOVL C01927 V=800.0 PL=0
MOVL C01928 V=800.0 PL=0
MOVL C01929 V=800.0 PL=0
MOVL C01930 V=800.0 PL=0
MOVL C01931 V=800.0 PL=0
MOVL C01932 V=800.0 PL=0
MOVL C01933 V=800.0 PL=0
MOVL C01934 V=800.0 PL=0
MOVL C01935 V=800.0 PL=0
MOVL C01936 V=800.0 PL=0
MOVL C01937 V=800.0 PL=0
MOVL C01938 V=800.0 PL=0
MOVL C01939 V=800.0 PL=0
MOVL C01940 V=800.0 PL=0
MOVL C01941 V=800.0 PL=0
MOVL C01942 V=800.0 PL=0
MOVL C01943 V=800.0 PL=0
MOVL C01944 V=800.0 PL=0
MOVL C01945 V=800.0 PL=0
MOVL C01946 V=800.0 PL=0
MOVL C01947 V=800.0 PL=0
MOVL C01948 V=800.0 PL=0
MOVL C01949 V=800.0 PL=0
MOVL C01950 V=800.0 PL=0
MOVL C01951 V=800.0 PL=0
MOVL C01952 V=800.0 PL=0
MOVL C01953 V=800.0 PL=0
MOVL C01954 V=800.0 PL=0
MOVL C01955 V=800.0 PL=0
MOVL C01956 V=800.0 PL=0
MOVL C01957 V=800.0 PL=0
MOVL C01958 V=800.0 PL=0
MOVL C01959 V=800.0 PL=0
MOVL C01960 V=800.0 PL=0
MOVL C01961 V=800.0 PL=0
MOVL C01962 V=800.0 PL=0
MOVL C01963 V=800.0 PL=0
MOVL C01964 V=800.0 PL=0
MOVL C01965 V=800.0 PL=0
MOVL C01966 V=800.0 PL=0
MOVL C01967 V=800.0 PL=0
MOVL C01968 V=800.0 PL=0
MOVL C01969 V=800.0 PL=0
MOVL C01970 V=800.0 PL=0
MOVL C01971 V=800.0 PL=0
MOVL C01972 V=800.0 PL=0
MOVL C01973 V=800.0 PL=0
MOVL C01974 V=800.0 PL=0
MOVL C01975 V=800.0 PL=0
MOVL C01976 V=800.0 PL=0
MOVL C01977 V=800.0 PL=0
MOVL C01978 V=800.0 PL=0
MOVL C01979 V=800.0 PL=0
MOVL C01980 V=800.0 PL=0
MOVL C01981 V=800.0 PL=0
MOVL C01982 V=800.0 PL=0
MOVL C01983 V=800.0 PL=0
MOVL C01984 V=800.0 PL=0
MOVL C01985 V=800.0 PL=0
MOVL C01986 V=800.0 PL=0
MOVL C01987 V=800.0 PL=0
MOVL C01988 V=800.0 PL=0
MOVL C01989 V=800.0 PL=0
MOVL C01990 V=800.0 PL=0
MOVL C01991 V=800.0 PL=0
MOVL C01992 V=800.0 PL=0
MOVL C01993 V=800.0 PL=0
MOVL C01994 V=800.0 PL=0
MOVL C01995 V=800.0 PL=0
MOVL C01996 V=800.0 PL=0
MOVL C01997 V=800.0 PL=0
MOVL C01998 V=800.0 PL=0
MOVL C01999 V=800.0 PL=0
MOVL C02000 V=800.0 PL=0
MOVL C02001 V=800.0 PL=0
MOVL C02002 V=800.0 PL=0
MOVL C02003 V=800.0 PL=0
MOVL C02004 V=800.0 PL=0
MOVL C02005 V=800.0 PL=0
MOVL C02006 V=800.0 PL=0
MOVL C02007 V=800.0 PL=0
MOVL C02008 V=800.0 PL=0
MOVL C02009 V=800.0 PL=0
MOVL C02010 V=800.0 PL=0
MOVL C02011 V=800.0 PL=0
MOVL C02012 V=800.0 PL=0
MOVL C02013 V=800.0 PL=0
MOVL C02014 V=800.0 PL=0
MOVL C02015 V=800.0 PL=0
MOVL C02016 V=800.0 PL=0
MOVL C02017 V=800.0 PL=0
MOVL C02018 V=800.0 PL=0
MOVL C02019 V=800.0 PL=0
MOVL C02020 V=800.0 PL=0
MOVL C02021 V=800.0 PL=0
MOVL C02022 V=800.0 PL=0
MOVL C02023 V=800.0 PL=0
MOVL C02024 V=800.0 PL=0
MOVL C02025 V=800.0 PL=0
MOVL C02026 V=800.0 PL=0
MOVL C02027 V=800.0 PL=0
MOVL C02028 V=800.0 PL=0
MOVL C02029 V=800.0 PL=0
MOVL C02030 V=800.0 PL=0
MOVL C02031 V=800.0 PL=0
MOVL C02032 V=800.0 PL=0
MOVL C02033 V=800.0 PL=0
MOVL C02034 V=800.0 PL=0
MOVL C02035 V=800.0 PL=0
MOVL C02036 V=800.0 PL=0
MOVL C02037 V=800.0 PL=0
MOVL C02038 V=800.0 PL=0
MOVL C02039 V=800.0 PL=0
MOVL C02040 V=800.0 PL=0
MOVL C02041 V=800.0 PL=0
MOVL C02042 V=800.0 PL=0
MOVL C02043 V=800.0 PL=0
MOVL C02044 V=800.0 PL=0
MOVL C02045 V=800.0 PL=0
MOVL C02046 V=800.0 PL=0
MOVL C02047 V=800.0 PL=0
MOVL C02048 V=800.0 PL=0
MOVL C02049 V=800.0 PL=0
MOVL C02050 V=800.0 PL=0
MOVL C02051 V=800.0 PL=0
MOVL C02052 V=800.0 PL=0
MOVL C02053 V=800.0 PL=0
MOVL C02054 V=800.0 PL=0
MOVL C02055 V=800.0 PL=0
MOVL C02056 V=800.0 PL=0
MOVL C02057 V=800.0 PL=0
MOVL C02058 V=800.0 PL=0
MOVL C02059 V=800.0 PL=0
MOVL C02060 V=800.0 PL=0
MOVL C02061 V=800.0 PL=0
MOVL C02062 V=800.0 PL=0
MOVL C02063 V=800.0 PL=0
MOVL C02064 V=800.0 PL=0
MOVL C02065 V=800.0 PL=0
MOVL C02066 V=800.0 PL=0
MOVL C02067 V=800.0 PL=0
MOVL C02068 V=800.0 PL=0
MOVL C02069 V=800.0 PL=0
MOVL C02070 V=800.0 PL=0
MOVL C02071 V=800.0 PL=0
MOVL C02072 V=800.0 PL=0
MOVL C02073 V=800.0 PL=0
MOVL C02074 V=800.0 PL=0
MOVL C02075 V=800.0 PL=0
MOVL C02076 V=800.0 PL=0
MOVL C02077 V=800.0 PL=0
MOVL C02078 V=800.0 PL=0
MOVL C02079 V=800.0 PL=0
MOVL C02080 V=800.0 PL=0
MOVL C02081 V=800.0 PL=0
MOVL C02082 V=800.0 PL=0
MOVL C02083 V=800.0 PL=0
MOVL C02084 V=800.0 PL=0
MOVL C02085 V=800.0 PL=0
MOVL C02086 V=800.0 PL=0
MOVL C02087 V=800.0 PL=0
MOVL C02088 V=800.0 PL=0
MOVL C02089 V=800.0 PL=0
MOVL C02090 V=800.0 PL=0
MOVL C02091 V=800.0 PL=0
MOVL C02092 V=800.0 PL=0
MOVL C02093 V=800.0 PL=0
MOVL C02094 V=800.0 PL=0
MOVL C02095 V=800.0 PL=0
MOVL C02096 V=800.0 PL=0
MOVL C02097 V=800.0 PL=0
MOVL C02098 V=800.0 PL=0
MOVL C02099 V=800.0 PL=0
MOVL C02100 V=800.0 PL=0
MOVL C02101 V=800.0 PL=0
MOVL C02102 V=800.0 PL=0
MOVL C02103 V=800.0 PL=0
MOVL C02104 V=800.0 PL=0
MOVL C02105 V=800.0 PL=0
MOVL C02106 V=800.0 PL=0
MOVL C02107 V=800.0 PL=0
MOVL C02108 V=800.0 PL=0
MOVL C02109 V=800.0 PL=0
MOVL C02110 V=800.0 PL=0
MOVL C02111 V=800.0 PL=0
MOVL C02112 V=800.0 PL=0
MOVL C02113 V=800.0 PL=0
MOVL C02114 V=800.0 PL=0
MOVL C02115 V=800.0 PL=0
MOVL C02116 V=800.0 PL=0
MOVL C02117 V=800.0 PL=0
MOVL C02118 V=800.0 PL=0
MOVL C02119 V=800.0 PL=0
MOVL C02120 V=800.0 PL=0
MOVL C02121 V=800.0 PL=0
MOVL C02122 V=800.0 PL=0
MOVL C02123 V=800.0 PL=0
MOVL C02124 V=800.0 PL=0
MOVL C02125 V=800.0 PL=0
MOVL C02126 V=800.0 PL=0
MOVL C02127 V=800.0 PL=0
MOVL C02128 V=800.0 PL=0
MOVL C02129 V=800.0 PL=0
MOVL C02130 V=800.0 PL=0
MOVL C02131 V=800.0 PL=0
MOVL C02132 V=800.0 PL=0
